LIN {X 0,Y 369.118,Z 198.507,A -85,B 0,C 180,E1 -12878.761,E2 -12878.761} C_VEL
LIN {X 0,Y 369.001,Z 198.517,A -85,B 0,C 180,E1 -12882.092,E2 -12882.092} C_VEL
LIN {X 0,Y 368.993,Z 198.519,A -85,B 0,C 180,E1 -12885.453,E2 -12885.453} C_VEL
LIN {X 0,Y 368.349,Z 198.603,A -85,B 0,C 180,E1 -12886.364,E2 -12886.364} C_VEL
LIN {X 0,Y 365.461,Z 198.96,A -85,B 0,C 180,E1 -12887.844,E2 -12887.844} C_VEL
LIN {X 0,Y 363.003,Z 199.268,A -85,B 0,C 180,E1 -12889.041,E2 -12889.041} C_VEL
LIN {X 0,Y 361.96,Z 199.395,A -85,B 0,C 180,E1 -12889.968,E2 -12889.968} C_VEL
LIN {X 0,Y 361.883,Z 199.405,A -85,B 0,C 180,E1 -12890.282,E2 -12890.282} C_VEL
LIN {X 0,Y 361.89,Z 199.404,A -85,B 0,C 180,E1 -12894.113,E2 -12894.113} C_VEL
LIN {X 0,Y 361.937,Z 199.403,A -85,B 0,C 180,E1 -12896.721,E2 -12896.721} C_VEL
LIN {X 0,Y 361.868,Z 199.409,A -85,B 0,C 180,E1 -12900.327,E2 -12900.327} C_VEL
LIN {X 0,Y 361.854,Z 199.411,A -85,B 0,C 180,E1 -12904.279,E2 -12904.279} C_VEL
LIN {X 0,Y 361.859,Z 199.407,A -85,B 0,C 180,E1 -12907.223,E2 -12907.223} C_VEL
LIN {X 0,Y 361.899,Z 199.405,A -85,B 0,C 180,E1 -12910.768,E2 -12910.768} C_VEL
LIN {X 0,Y 361.896,Z 199.408,A -85,B 0,C 180,E1 -12914.355,E2 -12914.355} C_VEL
LIN {X 0,Y 361.849,Z 199.408,A -85,B 0,C 180,E1 -12917.564,E2 -12917.564} C_VEL
LIN {X 0,Y 361.866,Z 199.406,A -85,B 0,C 180,E1 -12920.972,E2 -12920.972} C_VEL
LIN {X 0,Y 361.866,Z 199.408,A -85,B 0,C 180,E1 -12924.655,E2 -12924.655} C_VEL
LIN {X 0,Y 361.853,Z 199.412,A -85,B 0,C 180,E1 -12928.373,E2 -12928.373} C_VEL
LIN {X 0,Y 361.915,Z 199.405,A -85,B 0,C 180,E1 -12932.222,E2 -12932.222} C_VEL
LIN {X 0,Y 361.92,Z 199.4,A -85,B 0,C 180,E1 -12934.71,E2 -12934.71} C_VEL
LIN {X 0,Y 361.883,Z 199.407,A -85,B 0,C 180,E1 -12938.347,E2 -12938.347} C_VEL
LIN {X 0,Y 361.959,Z 199.4,A -85,B 0,C 180,E1 -12942.061,E2 -12942.061} C_VEL
LIN {X 0,Y 361.989,Z 199.395,A -85,B 0,C 180,E1 -12946.101,E2 -12946.101} C_VEL
LIN {X 0,Y 362.023,Z 199.392,A -85,B 0,C 180,E1 -12949.938,E2 -12949.938} C_VEL
LIN {X 0,Y 362.154,Z 199.372,A -85,B 0,C 180,E1 -12953.314,E2 -12953.314} C_VEL
LIN {X 0,Y 362.272,Z 199.361,A -85,B 0,C 180,E1 -12957.777,E2 -12957.777} C_VEL
LIN {X 0,Y 362.42,Z 199.34,A -85,B 0,C 180,E1 -12960.001,E2 -12960.001} C_VEL
LIN {X 0,Y 362.273,Z 199.356,A -85,B 0,C 180,E1 -12962.224,E2 -12962.224} C_VEL
LIN {X 0,Y 362.163,Z 199.369,A -85,B 0,C 180,E1 -12966.687,E2 -12966.687} C_VEL
LIN {X 0,Y 362.067,Z 199.382,A -85,B 0,C 180,E1 -12968.934,E2 -12968.934} C_VEL
LIN {X 0,Y 361.953,Z 199.395,A -85,B 0,C 180,E1 -12972.333,E2 -12972.333} C_VEL
LIN {X 0,Y 361.955,Z 199.395,A -85,B 0,C 180,E1 -12974.621,E2 -12974.621} C_VEL
LIN {X 0,Y 361.949,Z 199.396,A -85,B 0,C 180,E1 -12978.1,E2 -12978.1} C_VEL
LIN {X 0,Y 361.887,Z 199.406,A -85,B 0,C 180,E1 -12981.654,E2 -12981.654} C_VEL
LIN {X 0,Y 361.923,Z 199.405,A -85,B 0,C 180,E1 -12985.291,E2 -12985.291} C_VEL
LIN {X 0,Y 361.903,Z 199.403,A -85,B 0,C 180,E1 -12987.78,E2 -12987.78} C_VEL
LIN {X 0,Y 361.832,Z 199.412,A -85,B 0,C 180,E1 -12991.63,E2 -12991.63} C_VEL
LIN {X 0,Y 361.869,Z 199.409,A -85,B 0,C 180,E1 -12995.346,E2 -12995.346} C_VEL
LIN {X 0,Y 361.865,Z 199.412,A -85,B 0,C 180,E1 -12999.028,E2 -12999.028} C_VEL
LIN {X 0,Y 361.832,Z 199.415,A -85,B 0,C 180,E1 -13002.83,E2 -13002.83} C_VEL
LIN {X 0,Y 361.814,Z 199.412,A -85,B 0,C 180,E1 -13005.948,E2 -13005.948} C_VEL
LIN {X 0,Y 361.832,Z 199.413,A -85,B 0,C 180,E1 -13009.246,E2 -13009.246} C_VEL
LIN {X 0,Y 361.861,Z 199.412,A -85,B 0,C 180,E1 -13012.779,E2 -13012.779} C_VEL
LIN {X 0,Y 361.853,Z 199.412,A -85,B 0,C 180,E1 -13015.721,E2 -13015.721} C_VEL
LIN {X 0,Y 361.922,Z 199.576,A -85,B 0,C 180,E1 -13018.36,E2 -13018.36} C_VEL
LIN {X 0,Y 366.088,Z 217.855,A -85,B 0,C 180,E1 -13022.018,E2 -13022.018} C_VEL
LIN {X 0,Y 367.272,Z 224.486,A -85,B 0,C 180,E1 -13023.277,E2 -13023.277} C_VEL
LIN {X 0,Y 365.521,Z 242.961,A -85,B 0,C 180,E1 -13026.487,E2 -13026.487} C_VEL
LIN {X 0,Y 364.027,Z 261.035,A -85,B 0,C 180,E1 -13029.592,E2 -13029.592} C_VEL
LIN {X 0,Y 364.567,Z 267.895,A -85,B 0,C 180,E1 -13029.815,E2 -13029.815} C_VEL
LIN {X 0,Y 366.923,Z 292.032,A -85,B 0,C 180,E1 -13030.464,E2 -13030.464} C_VEL
LIN {X 0,Y 365.654,Z 367.753,A -85,B 0,C 180,E1 -13032.163,E2 -13032.163} C_VEL
LIN {X 0,Y 365.071,Z 380.038,A -85,B 0,C 180,E1 -13032.64,E2 -13032.64} C_VEL
LIN {X 0,Y 364.412,Z 392.244,A -85,B 0,C 180,E1 -13033.33,E2 -13033.33} C_VEL
LIN {X 0,Y 363.594,Z 404.788,A -85,B 0,C 180,E1 -13034.3,E2 -13034.3} C_VEL
LIN {X 0,Y 362.777,Z 415.954,A -85,B 0,C 180,E1 -13035.414,E2 -13035.414} C_VEL
LIN {X 0,Y 362.223,Z 424.979,A -85,B 0,C 180,E1 -13036.537,E2 -13036.537} C_VEL
LIN {X 0,Y 361.507,Z 434.174,A -85,B 0,C 180,E1 -13037.938,E2 -13037.938} C_VEL
LIN {X 0,Y 361.008,Z 443.11,A -85,B 0,C 180,E1 -13039.627,E2 -13039.627} C_VEL
LIN {X 0,Y 360.768,Z 450.158,A -85,B 0,C 180,E1 -13041.317,E2 -13041.317} C_VEL
LIN {X 0,Y 360.739,Z 456.564,A -85,B 0,C 180,E1 -13043.288,E2 -13043.288} C_VEL
LIN {X 0,Y 360.684,Z 460.629,A -85,B 0,C 180,E1 -13044.97,E2 -13044.97} C_VEL
LIN {X 0,Y 360.827,Z 463.562,A -85,B 0,C 180,E1 -13046.651,E2 -13046.651} C_VEL
LIN {X 0,Y 360.942,Z 464.906,A -85,B 0,C 180,E1 -13047.769,E2 -13047.769} C_VEL
LIN {X 0,Y 360.853,Z 465.795,A -85,B 0,C 180,E1 -13048.885,E2 -13048.885} C_VEL
LIN {X 0,Y 360.828,Z 466.258,A -85,B 0,C 180,E1 -13050.001,E2 -13050.001} C_VEL
LIN {X 0,Y 360.849,Z 466.244,A -85,B 0,C 180,E1 -13051.117,E2 -13051.117} C_VEL
LIN {X 0,Y 360.809,Z 465.799,A -85,B 0,C 180,E1 -13052.233,E2 -13052.233} C_VEL
LIN {X 0,Y 360.728,Z 464.934,A -85,B 0,C 180,E1 -13053.352,E2 -13053.352} C_VEL
LIN {X 0,Y 360.603,Z 463.587,A -85,B 0,C 180,E1 -13054.472,E2 -13054.472} C_VEL
LIN {X 0,Y 360.614,Z 460.433,A -85,B 0,C 180,E1 -13056.308,E2 -13056.308} C_VEL
LIN {X 0,Y 360.671,Z 456.84,A -85,B 0,C 180,E1 -13057.84,E2 -13057.84} C_VEL
LIN {X 0,Y 360.843,Z 451.756,A -85,B 0,C 180,E1 -13059.53,E2 -13059.53} C_VEL
LIN {X 0,Y 361.284,Z 445.363,A -85,B 0,C 180,E1 -13061.218,E2 -13061.218} C_VEL
LIN {X 0,Y 362.058,Z 437.426,A -85,B 0,C 180,E1 -13062.899,E2 -13062.899} C_VEL
LIN {X 0,Y 362.963,Z 429.132,A -85,B 0,C 180,E1 -13064.318,E2 -13064.318} C_VEL
LIN {X 0,Y 364.091,Z 418.285,A -85,B 0,C 180,E1 -13065.823,E2 -13065.823} C_VEL
LIN {X 0,Y 365.254,Z 408.426,A -85,B 0,C 180,E1 -13066.92,E2 -13066.92} C_VEL
LIN {X 0,Y 366.553,Z 395.984,A -85,B 0,C 180,E1 -13068.01,E2 -13068.01} C_VEL
LIN {X 0,Y 367.703,Z 383.82,A -85,B 0,C 180,E1 -13068.817,E2 -13068.817} C_VEL
LIN {X 0,Y 368.675,Z 370.254,A -85,B 0,C 180,E1 -13069.452,E2 -13069.452} C_VEL
LIN {X 0,Y 369.241,Z 356.669,A -85,B 0,C 180,E1 -13069.855,E2 -13069.855} C_VEL
LIN {X 0,Y 370.878,Z 292.289,A -85,B 0,C 180,E1 -13071.366,E2 -13071.366} C_VEL
LIN {X 0,Y 368.918,Z 273.49,A -85,B 0,C 180,E1 -13072.034,E2 -13072.034} C_VEL
LIN {X 0,Y 366.562,Z 258.445,A -85,B 0,C 180,E1 -13072.665,E2 -13072.665} C_VEL
LIN {X 0,Y 368.887,Z 236.241,A -85,B 0,C 180,E1 -13076.434,E2 -13076.434} C_VEL
LIN {X 0,Y 369.664,Z 228.641,A -85,B 0,C 180,E1 -13077.762,E2 -13077.762} C_VEL
LIN {X 0,Y 367.627,Z 218.97,A -85,B 0,C 180,E1 -13079.805,E2 -13079.805} C_VEL
LIN {X 0,Y 364.549,Z 207.813,A -85,B 0,C 180,E1 -13082.388,E2 -13082.388} C_VEL
LIN {X 0,Y 361.903,Z 199.531,A -85,B 0,C 180,E1 -13084.55,E2 -13084.55} C_VEL
LIN {X 0,Y 361.846,Z 199.412,A -85,B 0,C 180,E1 -13088.428,E2 -13088.428} C_VEL
LIN {X 0,Y 361.833,Z 199.413,A -85,B 0,C 180,E1 -13092.431,E2 -13092.431} C_VEL
LIN {X 0,Y 361.821,Z 199.413,A -85,B 0,C 180,E1 -13095.947,E2 -13095.947} C_VEL
LIN {X 0,Y 361.838,Z 199.413,A -85,B 0,C 180,E1 -13099.245,E2 -13099.245} C_VEL
LIN {X 0,Y 361.866,Z 199.409,A -85,B 0,C 180,E1 -13102.777,E2 -13102.777} C_VEL
LIN {X 0,Y 361.857,Z 199.409,A -85,B 0,C 180,E1 -13105.719,E2 -13105.719} C_VEL
LIN {X 0,Y 361.876,Z 199.408,A -85,B 0,C 180,E1 -13109.672,E2 -13109.672} C_VEL
LIN {X 0,Y 361.957,Z 199.397,A -85,B 0,C 180,E1 -13113.475,E2 -13113.475} C_VEL
LIN {X 0,Y 361.893,Z 199.403,A -85,B 0,C 180,E1 -13117.144,E2 -13117.144} C_VEL
LIN {X 0,Y 361.909,Z 199.403,A -85,B 0,C 180,E1 -13120.723,E2 -13120.723} C_VEL
LIN {X 0,Y 361.935,Z 199.401,A -85,B 0,C 180,E1 -13123.066,E2 -13123.066} C_VEL
LIN {X 0,Y 362.001,Z 199.394,A -85,B 0,C 180,E1 -13126.527,E2 -13126.527} C_VEL
LIN {X 0,Y 362.002,Z 199.394,A -85,B 0,C 180,E1 -13129.937,E2 -13129.937} C_VEL
LIN {X 0,Y 362.127,Z 199.581,A -85,B 0,C 180,E1 -13132.192,E2 -13132.192} C_VEL
LIN {X 0,Y 364.475,Z 207.695,A -85,B 0,C 180,E1 -13134.467,E2 -13134.467} C_VEL
LIN {X 0,Y 367.073,Z 217.573,A -85,B 0,C 180,E1 -13137.04,E2 -13137.04} C_VEL
LIN {X 0,Y 367.388,Z 220.859,A -85,B 0,C 180,E1 -13137.807,E2 -13137.807} C_VEL
LIN {X 0,Y 366.614,Z 232.738,A -85,B 0,C 180,E1 -13140.311,E2 -13140.311} C_VEL
LIN {X 0,Y 370.37,Z 248.389,A -85,B 0,C 180,E1 -13141.153,E2 -13141.153} C_VEL
LIN {X 0,Y 371.438,Z 253.878,A -85,B 0,C 180,E1 -13141.414,E2 -13141.414} C_VEL
LIN {X 0,Y 369.117,Z 317.897,A -85,B 0,C 180,E1 -13143.206,E2 -13143.206} C_VEL
LIN {X 0,Y 368.661,Z 330.151,A -85,B 0,C 180,E1 -13143.757,E2 -13143.757} C_VEL
LIN {X 0,Y 367.891,Z 342.582,A -85,B 0,C 180,E1 -13144.567,E2 -13144.567} C_VEL
LIN {X 0,Y 367.075,Z 353.098,A -85,B 0,C 180,E1 -13145.493,E2 -13145.493} C_VEL
LIN {X 0,Y 366.125,Z 363.059,A -85,B 0,C 180,E1 -13146.613,E2 -13146.613} C_VEL
LIN {X 0,Y 365.122,Z 372.767,A -85,B 0,C 180,E1 -13148.021,E2 -13148.021} C_VEL
LIN {X 0,Y 364.273,Z 379.966,A -85,B 0,C 180,E1 -13149.347,E2 -13149.347} C_VEL
LIN {X 0,Y 363.412,Z 386.564,A -85,B 0,C 180,E1 -13150.868,E2 -13150.868} C_VEL
LIN {X 0,Y 362.746,Z 391.42,A -85,B 0,C 180,E1 -13152.305,E2 -13152.305} C_VEL
LIN {X 0,Y 362.112,Z 395.64,A -85,B 0,C 180,E1 -13153.971,E2 -13153.971} C_VEL
LIN {X 0,Y 361.583,Z 398.748,A -85,B 0,C 180,E1 -13155.79,E2 -13155.79} C_VEL
LIN {X 0,Y 361.22,Z 400.374,A -85,B 0,C 180,E1 -13157.568,E2 -13157.568} C_VEL
LIN {X 0,Y 361.004,Z 400.698,A -85,B 0,C 180,E1 -13159.326,E2 -13159.326} C_VEL
LIN {X 0,Y 360.924,Z 399.948,A -85,B 0,C 180,E1 -13160.825,E2 -13160.825} C_VEL
LIN {X 0,Y 360.93,Z 399.056,A -85,B 0,C 180,E1 -13161.713,E2 -13161.713} C_VEL
LIN {X 0,Y 361.009,Z 397.344,A -85,B 0,C 180,E1 -13162.914,E2 -13162.914} C_VEL
LIN {X 0,Y 361.224,Z 393.503,A -85,B 0,C 180,E1 -13164.727,E2 -13164.727} C_VEL
LIN {X 0,Y 361.586,Z 387.777,A -85,B 0,C 180,E1 -13166.609,E2 -13166.609} C_VEL
LIN {X 0,Y 361.901,Z 381.824,A -85,B 0,C 180,E1 -13168.094,E2 -13168.094} C_VEL
LIN {X 0,Y 362.441,Z 373.721,A -85,B 0,C 180,E1 -13169.669,E2 -13169.669} C_VEL
LIN {X 0,Y 362.996,Z 364.815,A -85,B 0,C 180,E1 -13171.029,E2 -13171.029} C_VEL
LIN {X 0,Y 363.509,Z 355.694,A -85,B 0,C 180,E1 -13172.147,E2 -13172.147} C_VEL
LIN {X 0,Y 364.102,Z 344.601,A -85,B 0,C 180,E1 -13173.209,E2 -13173.209} C_VEL
LIN {X 0,Y 364.55,Z 332.719,A -85,B 0,C 180,E1 -13174.066,E2 -13174.066} C_VEL
LIN {X 0,Y 364.913,Z 321.208,A -85,B 0,C 180,E1 -13174.662,E2 -13174.662} C_VEL
LIN {X 0,Y 365.142,Z 308.779,A -85,B 0,C 180,E1 -13175.079,E2 -13175.079} C_VEL
LIN {X 0,Y 366.241,Z 249.047,A -85,B 0,C 180,E1 -13176.541,E2 -13176.541} C_VEL
LIN {X 0,Y 363.319,Z 230.123,A -85,B 0,C 180,E1 -13177.174,E2 -13177.174} C_VEL
LIN {X 0,Y 363.83,Z 216.259,A -85,B 0,C 180,E1 -13180.323,E2 -13180.323} C_VEL
LIN {X 0,Y 364.006,Z 210.426,A -85,B 0,C 180,E1 -13181.686,E2 -13181.686} C_VEL
LIN {X 0,Y 361.885,Z 199.568,A -85,B 0,C 180,E1 -13184.454,E2 -13184.454} C_VEL
LIN {X 0,Y 361.835,Z 199.415,A -85,B 0,C 180,E1 -13187.567,E2 -13187.567} C_VEL
LIN {X 0,Y 361.867,Z 199.406,A -85,B 0,C 180,E1 -13190.973,E2 -13190.973} C_VEL
LIN {X 0,Y 361.873,Z 199.405,A -85,B 0,C 180,E1 -13194.655,E2 -13194.655} C_VEL
LIN {X 0,Y 361.838,Z 199.41,A -85,B 0,C 180,E1 -13198.37,E2 -13198.37} C_VEL
LIN {X 0,Y 361.899,Z 199.403,A -85,B 0,C 180,E1 -13200.955,E2 -13200.955} C_VEL
LIN {X 0,Y 361.953,Z 199.401,A -85,B 0,C 180,E1 -13203.474,E2 -13203.474} C_VEL
LIN {X 0,Y 361.889,Z 199.406,A -85,B 0,C 180,E1 -13207.144,E2 -13207.144} C_VEL
LIN {X 0,Y 361.919,Z 199.4,A -85,B 0,C 180,E1 -13210.723,E2 -13210.723} C_VEL
LIN {X 0,Y 361.944,Z 199.396,A -85,B 0,C 180,E1 -13214.225,E2 -13214.225} C_VEL
LIN {X 0,Y 361.997,Z 199.39,A -85,B 0,C 180,E1 -13216.527,E2 -13216.527} C_VEL
LIN {X 0,Y 362.029,Z 199.386,A -85,B 0,C 180,E1 -13219.937,E2 -13219.937} C_VEL
LIN {X 0,Y 362.149,Z 199.371,A -85,B 0,C 180,E1 -13222.192,E2 -13222.192} C_VEL
LIN {X 0,Y 362.116,Z 199.375,A -85,B 0,C 180,E1 -13224.43,E2 -13224.43} C_VEL
LIN {X 0,Y 362.28,Z 199.355,A -85,B 0,C 180,E1 -13227.776,E2 -13227.776} C_VEL
LIN {X 0,Y 362.425,Z 199.336,A -85,B 0,C 180,E1 -13229.999,E2 -13229.999} C_VEL
LIN {X 0,Y 362.28,Z 199.354,A -85,B 0,C 180,E1 -13232.223,E2 -13232.223} C_VEL
LIN {X 0,Y 362.157,Z 199.373,A -85,B 0,C 180,E1 -13236.686,E2 -13236.686} C_VEL
LIN {X 0,Y 362.028,Z 199.386,A -85,B 0,C 180,E1 -13240.061,E2 -13240.061} C_VEL
LIN {X 0,Y 361.993,Z 199.39,A -85,B 0,C 180,E1 -13243.898,E2 -13243.898} C_VEL
LIN {X 0,Y 361.962,Z 199.394,A -85,B 0,C 180,E1 -13247.938,E2 -13247.938} C_VEL
LIN {X 0,Y 361.883,Z 199.405,A -85,B 0,C 180,E1 -13250.282,E2 -13250.282} C_VEL
LIN {X 0,Y 361.233,Z 199.492,A -85,B 0,C 180,E1 -13251.211,E2 -13251.211} C_VEL
LIN {X 0,Y 358.371,Z 199.85,A -85,B 0,C 180,E1 -13252.722,E2 -13252.722} C_VEL
LIN {X 0,Y 355.949,Z 200.148,A -85,B 0,C 180,E1 -13253.944,E2 -13253.944} C_VEL
LIN {X 0,Y 354.927,Z 200.274,A -85,B 0,C 180,E1 -13254.89,E2 -13254.89} C_VEL
LIN {X 0,Y 354.854,Z 200.279,A -85,B 0,C 180,E1 -13255.211,E2 -13255.211} C_VEL
LIN {X 0,Y 354.845,Z 200.284,A -85,B 0,C 180,E1 -13258.38,E2 -13258.38} C_VEL
LIN {X 0,Y 354.787,Z 200.288,A -85,B 0,C 180,E1 -13261.594,E2 -13261.594} C_VEL
LIN {X 0,Y 354.81,Z 200.286,A -85,B 0,C 180,E1 -13265.058,E2 -13265.058} C_VEL
LIN {X 0,Y 354.801,Z 200.287,A -85,B 0,C 180,E1 -13267.882,E2 -13267.882} C_VEL
LIN {X 0,Y 354.833,Z 200.282,A -85,B 0,C 180,E1 -13271.181,E2 -13271.181} C_VEL
LIN {X 0,Y 354.85,Z 200.285,A -85,B 0,C 180,E1 -13274.521,E2 -13274.521} C_VEL
LIN {X 0,Y 354.806,Z 200.286,A -85,B 0,C 180,E1 -13277.665,E2 -13277.665} C_VEL
LIN {X 0,Y 354.829,Z 200.285,A -85,B 0,C 180,E1 -13280.669,E2 -13280.669} C_VEL
LIN {X 0,Y 354.814,Z 200.29,A -85,B 0,C 180,E1 -13284.3,E2 -13284.3} C_VEL
LIN {X 0,Y 354.791,Z 200.289,A -85,B 0,C 180,E1 -13287.668,E2 -13287.668} C_VEL
LIN {X 0,Y 354.861,Z 200.28,A -85,B 0,C 180,E1 -13290.621,E2 -13290.621} C_VEL
LIN {X 0,Y 354.891,Z 200.28,A -85,B 0,C 180,E1 -13294.173,E2 -13294.173} C_VEL
LIN {X 0,Y 354.826,Z 200.288,A -85,B 0,C 180,E1 -13297.894,E2 -13297.894} C_VEL
LIN {X 0,Y 354.915,Z 200.277,A -85,B 0,C 180,E1 -13301.891,E2 -13301.891} C_VEL
LIN {X 0,Y 354.935,Z 200.275,A -85,B 0,C 180,E1 -13305.981,E2 -13305.981} C_VEL
LIN {X 0,Y 354.97,Z 200.27,A -85,B 0,C 180,E1 -13309.736,E2 -13309.736} C_VEL
LIN {X 0,Y 355.118,Z 200.247,A -85,B 0,C 180,E1 -13313.181,E2 -13313.181} C_VEL
LIN {X 0,Y 355.235,Z 200.238,A -85,B 0,C 180,E1 -13317.733,E2 -13317.733} C_VEL
LIN {X 0,Y 355.389,Z 200.216,A -85,B 0,C 180,E1 -13320.001,E2 -13320.001} C_VEL
LIN {X 0,Y 355.236,Z 200.233,A -85,B 0,C 180,E1 -13322.268,E2 -13322.268} C_VEL
LIN {X 0,Y 355.129,Z 200.245,A -85,B 0,C 180,E1 -13326.82,E2 -13326.82} C_VEL
LIN {X 0,Y 355.008,Z 200.262,A -85,B 0,C 180,E1 -13329.113,E2 -13329.113} C_VEL
LIN {X 0,Y 354.914,Z 200.272,A -85,B 0,C 180,E1 -13332.582,E2 -13332.582} C_VEL
LIN {X 0,Y 354.883,Z 200.276,A -85,B 0,C 180,E1 -13336.097,E2 -13336.097} C_VEL
LIN {X 0,Y 354.895,Z 200.274,A -85,B 0,C 180,E1 -13338.473,E2 -13338.473} C_VEL
LIN {X 0,Y 354.83,Z 200.283,A -85,B 0,C 180,E1 -13342.107,E2 -13342.107} C_VEL
LIN {X 0,Y 354.893,Z 200.276,A -85,B 0,C 180,E1 -13345.828,E2 -13345.828} C_VEL
LIN {X 0,Y 354.812,Z 200.286,A -85,B 0,C 180,E1 -13349.683,E2 -13349.683} C_VEL
LIN {X 0,Y 354.801,Z 200.287,A -85,B 0,C 180,E1 -13353.703,E2 -13353.703} C_VEL
LIN {X 0,Y 354.793,Z 200.288,A -85,B 0,C 180,E1 -13356.461,E2 -13356.461} C_VEL
LIN {X 0,Y 354.82,Z 200.286,A -85,B 0,C 180,E1 -13359.425,E2 -13359.425} C_VEL
LIN {X 0,Y 354.784,Z 200.293,A -85,B 0,C 180,E1 -13362.868,E2 -13362.868} C_VEL
LIN {X 0,Y 354.763,Z 200.291,A -85,B 0,C 180,E1 -13366.105,E2 -13366.105} C_VEL
LIN {X 0,Y 354.784,Z 200.291,A -85,B 0,C 180,E1 -13369.18,E2 -13369.18} C_VEL
LIN {X 0,Y 354.804,Z 200.287,A -85,B 0,C 180,E1 -13372.404,E2 -13372.404} C_VEL
LIN {X 0,Y 354.81,Z 200.291,A -85,B 0,C 180,E1 -13374.942,E2 -13374.942} C_VEL
LIN {X 0,Y 354.864,Z 200.477,A -85,B 0,C 180,E1 -13378.052,E2 -13378.052} C_VEL
LIN {X 0,Y 359.007,Z 218.586,A -85,B 0,C 180,E1 -13381.756,E2 -13381.756} C_VEL
LIN {X 0,Y 360.296,Z 225.133,A -85,B 0,C 180,E1 -13383.032,E2 -13383.032} C_VEL
LIN {X 0,Y 359.033,Z 238.587,A -85,B 0,C 180,E1 -13385.421,E2 -13385.421} C_VEL
LIN {X 0,Y 357.085,Z 260.763,A -85,B 0,C 180,E1 -13389.319,E2 -13389.319} C_VEL
LIN {X 0,Y 358.098,Z 273.042,A -85,B 0,C 180,E1 -13389.692,E2 -13389.692} C_VEL
LIN {X 0,Y 359.973,Z 293.475,A -85,B 0,C 180,E1 -13390.248,E2 -13390.248} C_VEL
LIN {X 0,Y 358.736,Z 366.518,A -85,B 0,C 180,E1 -13391.918,E2 -13391.918} C_VEL
LIN {X 0,Y 358.104,Z 379.758,A -85,B 0,C 180,E1 -13392.439,E2 -13392.439} C_VEL
LIN {X 0,Y 357.408,Z 391.868,A -85,B 0,C 180,E1 -13393.141,E2 -13393.141} C_VEL
LIN {X 0,Y 356.591,Z 404.377,A -85,B 0,C 180,E1 -13394.131,E2 -13394.131} C_VEL
LIN {X 0,Y 355.788,Z 415.287,A -85,B 0,C 180,E1 -13395.241,E2 -13395.241} C_VEL
LIN {X 0,Y 355.164,Z 424.502,A -85,B 0,C 180,E1 -13396.41,E2 -13396.41} C_VEL
LIN {X 0,Y 354.4,Z 434.514,A -85,B 0,C 180,E1 -13397.983,E2 -13397.983} C_VEL
LIN {X 0,Y 353.971,Z 441.921,A -85,B 0,C 180,E1 -13399.418,E2 -13399.418} C_VEL
LIN {X 0,Y 353.683,Z 449.1,A -85,B 0,C 180,E1 -13401.142,E2 -13401.142} C_VEL
LIN {X 0,Y 353.673,Z 453.943,A -85,B 0,C 180,E1 -13402.58,E2 -13402.58} C_VEL
LIN {X 0,Y 353.694,Z 458.499,A -85,B 0,C 180,E1 -13404.299,E2 -13404.299} C_VEL
LIN {X 0,Y 353.598,Z 460.845,A -85,B 0,C 180,E1 -13405.441,E2 -13405.441} C_VEL
LIN {X 0,Y 353.761,Z 462.754,A -85,B 0,C 180,E1 -13406.584,E2 -13406.584} C_VEL
LIN {X 0,Y 353.893,Z 464.14,A -85,B 0,C 180,E1 -13407.725,E2 -13407.725} C_VEL
LIN {X 0,Y 353.808,Z 465.058,A -85,B 0,C 180,E1 -13408.863,E2 -13408.863} C_VEL
LIN {X 0,Y 353.78,Z 465.554,A -85,B 0,C 180,E1 -13410.001,E2 -13410.001} C_VEL
LIN {X 0,Y 353.8,Z 465.581,A -85,B 0,C 180,E1 -13411.139,E2 -13411.139} C_VEL
LIN {X 0,Y 353.737,Z 465.159,A -85,B 0,C 180,E1 -13412.278,E2 -13412.278} C_VEL
LIN {X 0,Y 353.632,Z 464.317,A -85,B 0,C 180,E1 -13413.419,E2 -13413.419} C_VEL
LIN {X 0,Y 353.526,Z 463.026,A -85,B 0,C 180,E1 -13414.562,E2 -13414.562} C_VEL
LIN {X 0,Y 353.518,Z 460.257,A -85,B 0,C 180,E1 -13416.271,E2 -13416.271} C_VEL
LIN {X 0,Y 353.571,Z 456.381,A -85,B 0,C 180,E1 -13417.999,E2 -13417.999} C_VEL
LIN {X 0,Y 353.787,Z 451.35,A -85,B 0,C 180,E1 -13419.722,E2 -13419.722} C_VEL
LIN {X 0,Y 354.292,Z 445.009,A -85,B 0,C 180,E1 -13421.442,E2 -13421.442} C_VEL
LIN {X 0,Y 355.085,Z 437.16,A -85,B 0,C 180,E1 -13423.157,E2 -13423.157} C_VEL
LIN {X 0,Y 356.144,Z 427.942,A -85,B 0,C 180,E1 -13424.771,E2 -13424.771} C_VEL
LIN {X 0,Y 357.25,Z 418.332,A -85,B 0,C 180,E1 -13426.134,E2 -13426.134} C_VEL
LIN {X 0,Y 358.494,Z 408.625,A -85,B 0,C 180,E1 -13427.249,E2 -13427.249} C_VEL
LIN {X 0,Y 359.685,Z 398.191,A -85,B 0,C 180,E1 -13428.218,E2 -13428.218} C_VEL
LIN {X 0,Y 360.894,Z 385.711,A -85,B 0,C 180,E1 -13429.112,E2 -13429.112} C_VEL
LIN {X 0,Y 361.962,Z 373.429,A -85,B 0,C 180,E1 -13429.754,E2 -13429.754} C_VEL
LIN {X 0,Y 362.61,Z 360.881,A -85,B 0,C 180,E1 -13430.197,E2 -13430.197} C_VEL
LIN {X 0,Y 364.548,Z 293.153,A -85,B 0,C 180,E1 -13431.846,E2 -13431.846} C_VEL
LIN {X 0,Y 362.577,Z 274.319,A -85,B 0,C 180,E1 -13432.535,E2 -13432.535} C_VEL
LIN {X 0,Y 360.02,Z 258.245,A -85,B 0,C 180,E1 -13433.232,E2 -13433.232} C_VEL
LIN {X 0,Y 362.35,Z 237.307,A -85,B 0,C 180,E1 -13436.848,E2 -13436.848} C_VEL
LIN {X 0,Y 363.076,Z 230.876,A -85,B 0,C 180,E1 -13437.993,E2 -13437.993} C_VEL
LIN {X 0,Y 361.091,Z 221.299,A -85,B 0,C 180,E1 -13440.078,E2 -13440.078} C_VEL
LIN {X 0,Y 358.056,Z 210.158,A -85,B 0,C 180,E1 -13442.745,E2 -13442.745} C_VEL
LIN {X 0,Y 354.865,Z 200.481,A -85,B 0,C 180,E1 -13445.373,E2 -13445.373} C_VEL
LIN {X 0,Y 354.797,Z 200.29,A -85,B 0,C 180,E1 -13447.884,E2 -13447.884} C_VEL
LIN {X 0,Y 354.774,Z 200.293,A -85,B 0,C 180,E1 -13451.168,E2 -13451.168} C_VEL
LIN {X 0,Y 354.766,Z 200.292,A -85,B 0,C 180,E1 -13454.506,E2 -13454.506} C_VEL
LIN {X 0,Y 354.797,Z 200.288,A -85,B 0,C 180,E1 -13457.662,E2 -13457.662} C_VEL
LIN {X 0,Y 354.819,Z 200.286,A -85,B 0,C 180,E1 -13460.666,E2 -13460.666} C_VEL
LIN {X 0,Y 354.825,Z 200.283,A -85,B 0,C 180,E1 -13464.301,E2 -13464.301} C_VEL
LIN {X 0,Y 354.79,Z 200.29,A -85,B 0,C 180,E1 -13467.666,E2 -13467.666} C_VEL
LIN {X 0,Y 354.85,Z 200.284,A -85,B 0,C 180,E1 -13471.618,E2 -13471.618} C_VEL
LIN {X 0,Y 354.902,Z 200.278,A -85,B 0,C 180,E1 -13474.172,E2 -13474.172} C_VEL
LIN {X 0,Y 354.838,Z 200.284,A -85,B 0,C 180,E1 -13477.894,E2 -13477.894} C_VEL
LIN {X 0,Y 354.925,Z 200.275,A -85,B 0,C 180,E1 -13481.891,E2 -13481.891} C_VEL
LIN {X 0,Y 354.945,Z 200.271,A -85,B 0,C 180,E1 -13485.981,E2 -13485.981} C_VEL
LIN {X 0,Y 354.958,Z 200.272,A -85,B 0,C 180,E1 -13489.735,E2 -13489.735} C_VEL
LIN {X 0,Y 355.062,Z 200.476,A -85,B 0,C 180,E1 -13491.348,E2 -13491.348} C_VEL
LIN {X 0,Y 357.879,Z 209.797,A -85,B 0,C 180,E1 -13494.082,E2 -13494.082} C_VEL
LIN {X 0,Y 360.579,Z 220.271,A -85,B 0,C 180,E1 -13496.887,E2 -13496.887} C_VEL
LIN {X 0,Y 360.761,Z 223.994,A -85,B 0,C 180,E1 -13497.767,E2 -13497.767} C_VEL
LIN {X 0,Y 360.124,Z 233.131,A -85,B 0,C 180,E1 -13499.72,E2 -13499.72} C_VEL
LIN {X 0,Y 363.944,Z 248.948,A -85,B 0,C 180,E1 -13500.622,E2 -13500.622} C_VEL
LIN {X 0,Y 365.125,Z 255.392,A -85,B 0,C 180,E1 -13500.93,E2 -13500.93} C_VEL
LIN {X 0,Y 362.685,Z 318.346,A -85,B 0,C 180,E1 -13502.741,E2 -13502.741} C_VEL
LIN {X 0,Y 362.171,Z 331.157,A -85,B 0,C 180,E1 -13503.337,E2 -13503.337} C_VEL
LIN {X 0,Y 361.453,Z 341.836,A -85,B 0,C 180,E1 -13504.041,E2 -13504.041} C_VEL
LIN {X 0,Y 360.535,Z 353.165,A -85,B 0,C 180,E1 -13505.03,E2 -13505.03} C_VEL
LIN {X 0,Y 359.568,Z 363.24,A -85,B 0,C 180,E1 -13506.171,E2 -13506.171} C_VEL
LIN {X 0,Y 358.673,Z 371.286,A -85,B 0,C 180,E1 -13507.317,E2 -13507.317} C_VEL
LIN {X 0,Y 357.637,Z 379.443,A -85,B 0,C 180,E1 -13508.759,E2 -13508.759} C_VEL
LIN {X 0,Y 356.747,Z 385.898,A -85,B 0,C 180,E1 -13510.212,E2 -13510.212} C_VEL
LIN {X 0,Y 355.869,Z 391.934,A -85,B 0,C 180,E1 -13511.967,E2 -13511.967} C_VEL
LIN {X 0,Y 355.182,Z 396.327,A -85,B 0,C 180,E1 -13513.735,E2 -13513.735} C_VEL
LIN {X 0,Y 354.768,Z 398.491,A -85,B 0,C 180,E1 -13514.923,E2 -13514.923} C_VEL
LIN {X 0,Y 354.463,Z 400.06,A -85,B 0,C 180,E1 -13516.115,E2 -13516.115} C_VEL
LIN {X 0,Y 354.136,Z 401.228,A -85,B 0,C 180,E1 -13517.714,E2 -13517.714} C_VEL
LIN {X 0,Y 353.899,Z 401.232,A -85,B 0,C 180,E1 -13519.73,E2 -13519.73} C_VEL
LIN {X 0,Y 353.847,Z 400.386,A -85,B 0,C 180,E1 -13521.012,E2 -13521.012} C_VEL
LIN {X 0,Y 353.939,Z 398.155,A -85,B 0,C 180,E1 -13522.78,E2 -13522.78} C_VEL
LIN {X 0,Y 354.159,Z 394.364,A -85,B 0,C 180,E1 -13524.627,E2 -13524.627} C_VEL
LIN {X 0,Y 354.474,Z 389.305,A -85,B 0,C 180,E1 -13526.374,E2 -13526.374} C_VEL
LIN {X 0,Y 354.818,Z 382.832,A -85,B 0,C 180,E1 -13528.061,E2 -13528.061} C_VEL
LIN {X 0,Y 355.347,Z 375.023,A -85,B 0,C 180,E1 -13529.633,E2 -13529.633} C_VEL
LIN {X 0,Y 355.912,Z 366.069,A -85,B 0,C 180,E1 -13531.055,E2 -13531.055} C_VEL
LIN {X 0,Y 356.526,Z 355.954,A -85,B 0,C 180,E1 -13532.323,E2 -13532.323} C_VEL
LIN {X 0,Y 357.136,Z 344.457,A -85,B 0,C 180,E1 -13533.435,E2 -13533.435} C_VEL
LIN {X 0,Y 357.609,Z 332.677,A -85,B 0,C 180,E1 -13534.288,E2 -13534.288} C_VEL
LIN {X 0,Y 357.945,Z 321.353,A -85,B 0,C 180,E1 -13534.878,E2 -13534.878} C_VEL
LIN {X 0,Y 358.183,Z 308.816,A -85,B 0,C 180,E1 -13535.303,E2 -13535.303} C_VEL
LIN {X 0,Y 359.3,Z 249.557,A -85,B 0,C 180,E1 -13536.79,E2 -13536.79} C_VEL
LIN {X 0,Y 356.372,Z 230.631,A -85,B 0,C 180,E1 -13537.413,E2 -13537.413} C_VEL
LIN {X 0,Y 356.673,Z 223.132,A -85,B 0,C 180,E1 -13539.089,E2 -13539.089} C_VEL
LIN {X 0,Y 357.1,Z 212.462,A -85,B 0,C 180,E1 -13541.593,E2 -13541.593} C_VEL
LIN {X 0,Y 355.151,Z 201.926,A -85,B 0,C 180,E1 -13544.263,E2 -13544.263} C_VEL
LIN {X 0,Y 354.823,Z 200.341,A -85,B 0,C 180,E1 -13544.753,E2 -13544.753} C_VEL
LIN {X 0,Y 354.793,Z 200.293,A -85,B 0,C 180,E1 -13547.662,E2 -13547.662} C_VEL
LIN {X 0,Y 354.814,Z 200.284,A -85,B 0,C 180,E1 -13550.665,E2 -13550.665} C_VEL
LIN {X 0,Y 354.82,Z 200.284,A -85,B 0,C 180,E1 -13554.3,E2 -13554.3} C_VEL
LIN {X 0,Y 354.788,Z 200.293,A -85,B 0,C 180,E1 -13557.666,E2 -13557.666} C_VEL
LIN {X 0,Y 354.867,Z 200.278,A -85,B 0,C 180,E1 -13560.621,E2 -13560.621} C_VEL
LIN {X 0,Y 354.898,Z 200.274,A -85,B 0,C 180,E1 -13564.172,E2 -13564.172} C_VEL
LIN {X 0,Y 354.833,Z 200.284,A -85,B 0,C 180,E1 -13567.893,E2 -13567.893} C_VEL
LIN {X 0,Y 354.921,Z 200.272,A -85,B 0,C 180,E1 -13571.891,E2 -13571.891} C_VEL
LIN {X 0,Y 354.941,Z 200.269,A -85,B 0,C 180,E1 -13575.98,E2 -13575.98} C_VEL
LIN {X 0,Y 354.976,Z 200.266,A -85,B 0,C 180,E1 -13579.735,E2 -13579.735} C_VEL
LIN {X 0,Y 355.112,Z 200.247,A -85,B 0,C 180,E1 -13582.036,E2 -13582.036} C_VEL
LIN {X 0,Y 355.091,Z 200.25,A -85,B 0,C 180,E1 -13584.32,E2 -13584.32} C_VEL
LIN {X 0,Y 355.243,Z 200.232,A -85,B 0,C 180,E1 -13587.732,E2 -13587.732} C_VEL
LIN {X 0,Y 355.395,Z 200.212,A -85,B 0,C 180,E1 -13589.999,E2 -13589.999} C_VEL
LIN {X 0,Y 355.243,Z 200.231,A -85,B 0,C 180,E1 -13592.267,E2 -13592.267} C_VEL
LIN {X 0,Y 355.122,Z 200.251,A -85,B 0,C 180,E1 -13596.819,E2 -13596.819} C_VEL
LIN {X 0,Y 354.974,Z 200.265,A -85,B 0,C 180,E1 -13600.263,E2 -13600.263} C_VEL
LIN {X 0,Y 354.938,Z 200.269,A -85,B 0,C 180,E1 -13604.018,E2 -13604.018} C_VEL
LIN {X 0,Y 354.918,Z 200.272,A -85,B 0,C 180,E1 -13608.108,E2 -13608.108} C_VEL
LIN {X 0,Y 354.83,Z 200.283,A -85,B 0,C 180,E1 -13612.105,E2 -13612.105} C_VEL
LIN {X 0,Y 354.854,Z 200.279,A -85,B 0,C 180,E1 -13615.211,E2 -13615.211} C_VEL
LIN {X 0,Y 354.214,Z 200.362,A -85,B 0,C 180,E1 -13616.157,E2 -13616.157} C_VEL
LIN {X 0,Y 351.364,Z 200.714,A -85,B 0,C 180,E1 -13617.696,E2 -13617.696} C_VEL
LIN {X 0,Y 348.922,Z 201.021,A -85,B 0,C 180,E1 -13618.942,E2 -13618.942} C_VEL
LIN {X 0,Y 347.856,Z 201.152,A -85,B 0,C 180,E1 -13619.906,E2 -13619.906} C_VEL
LIN {X 0,Y 347.762,Z 201.165,A -85,B 0,C 180,E1 -13620.233,E2 -13620.233} C_VEL
LIN {X 0,Y 347.742,Z 201.167,A -85,B 0,C 180,E1 -13624.043,E2 -13624.043} C_VEL
LIN {X 0,Y 347.757,Z 201.164,A -85,B 0,C 180,E1 -13627.32,E2 -13627.32} C_VEL
LIN {X 0,Y 347.787,Z 201.164,A -85,B 0,C 180,E1 -13630.288,E2 -13630.288} C_VEL
LIN {X 0,Y 347.776,Z 201.161,A -85,B 0,C 180,E1 -13633.398,E2 -13633.398} C_VEL
LIN {X 0,Y 347.762,Z 201.166,A -85,B 0,C 180,E1 -13636.678,E2 -13636.678} C_VEL
LIN {X 0,Y 347.75,Z 201.169,A -85,B 0,C 180,E1 -13640.171,E2 -13640.171} C_VEL
LIN {X 0,Y 347.758,Z 201.165,A -85,B 0,C 180,E1 -13642.68,E2 -13642.68} C_VEL
LIN {X 0,Y 347.74,Z 201.169,A -85,B 0,C 180,E1 -13645.956,E2 -13645.956} C_VEL
LIN {X 0,Y 347.764,Z 201.164,A -85,B 0,C 180,E1 -13649.654,E2 -13649.654} C_VEL
LIN {X 0,Y 347.823,Z 201.157,A -85,B 0,C 180,E1 -13653.608,E2 -13653.608} C_VEL
LIN {X 0,Y 347.78,Z 201.166,A -85,B 0,C 180,E1 -13656.162,E2 -13656.162} C_VEL
LIN {X 0,Y 347.809,Z 201.162,A -85,B 0,C 180,E1 -13659.91,E2 -13659.91} C_VEL
LIN {X 0,Y 347.859,Z 201.153,A -85,B 0,C 180,E1 -13662.359,E2 -13662.359} C_VEL
LIN {X 0,Y 347.889,Z 201.152,A -85,B 0,C 180,E1 -13665.971,E2 -13665.971} C_VEL
LIN {X 0,Y 347.921,Z 201.146,A -85,B 0,C 180,E1 -13669.526,E2 -13669.526} C_VEL
LIN {X 0,Y 348.084,Z 201.123,A -85,B 0,C 180,E1 -13673.042,E2 -13673.042} C_VEL
LIN {X 0,Y 348.198,Z 201.115,A -85,B 0,C 180,E1 -13677.687,E2 -13677.687} C_VEL
LIN {X 0,Y 348.338,Z 201.094,A -85,B 0,C 180,E1 -13680.001,E2 -13680.001} C_VEL
LIN {X 0,Y 348.198,Z 201.109,A -85,B 0,C 180,E1 -13682.314,E2 -13682.314} C_VEL
LIN {X 0,Y 348.098,Z 201.122,A -85,B 0,C 180,E1 -13686.958,E2 -13686.958} C_VEL
LIN {X 0,Y 347.96,Z 201.142,A -85,B 0,C 180,E1 -13689.299,E2 -13689.299} C_VEL
LIN {X 0,Y 347.883,Z 201.149,A -85,B 0,C 180,E1 -13692.84,E2 -13692.84} C_VEL
LIN {X 0,Y 347.832,Z 201.154,A -85,B 0,C 180,E1 -13696.432,E2 -13696.432} C_VEL
LIN {X 0,Y 347.845,Z 201.154,A -85,B 0,C 180,E1 -13698.861,E2 -13698.861} C_VEL
LIN {X 0,Y 347.769,Z 201.162,A -85,B 0,C 180,E1 -13702.58,E2 -13702.58} C_VEL
LIN {X 0,Y 347.807,Z 201.162,A -85,B 0,C 180,E1 -13705.109,E2 -13705.109} C_VEL
LIN {X 0,Y 347.803,Z 201.16,A -85,B 0,C 180,E1 -13707.695,E2 -13707.695} C_VEL
LIN {X 0,Y 347.744,Z 201.165,A -85,B 0,C 180,E1 -13710.349,E2 -13710.349} C_VEL
LIN {X 0,Y 347.744,Z 201.165,A -85,B 0,C 180,E1 -13714.045,E2 -13714.045} C_VEL
LIN {X 0,Y 347.757,Z 201.167,A -85,B 0,C 180,E1 -13717.322,E2 -13717.322} C_VEL
LIN {X 0,Y 347.728,Z 201.167,A -85,B 0,C 180,E1 -13720.298,E2 -13720.298} C_VEL
LIN {X 0,Y 347.719,Z 201.17,A -85,B 0,C 180,E1 -13723.409,E2 -13723.409} C_VEL
LIN {X 0,Y 347.722,Z 201.171,A -85,B 0,C 180,E1 -13726.688,E2 -13726.688} C_VEL
LIN {X 0,Y 347.744,Z 201.166,A -85,B 0,C 180,E1 -13730.174,E2 -13730.174} C_VEL
LIN {X 0,Y 347.759,Z 201.168,A -85,B 0,C 180,E1 -13732.68,E2 -13732.68} C_VEL
LIN {X 0,Y 347.747,Z 201.17,A -85,B 0,C 180,E1 -13735.957,E2 -13735.957} C_VEL
LIN {X 0,Y 347.827,Z 201.397,A -85,B 0,C 180,E1 -13737.745,E2 -13737.745} C_VEL
LIN {X 0,Y 351.767,Z 218.626,A -85,B 0,C 180,E1 -13741.349,E2 -13741.349} C_VEL
LIN {X 0,Y 353.25,Z 225.736,A -85,B 0,C 180,E1 -13742.769,E2 -13742.769} C_VEL
LIN {X 0,Y 352.826,Z 232.502,A -85,B 0,C 180,E1 -13744.011,E2 -13744.011} C_VEL
LIN {X 0,Y 350.526,Z 255.91,A -85,B 0,C 180,E1 -13748.229,E2 -13748.229} C_VEL
LIN {X 0,Y 350.153,Z 260.979,A -85,B 0,C 180,E1 -13749.076,E2 -13749.076} C_VEL
LIN {X 0,Y 353.071,Z 293.175,A -85,B 0,C 180,E1 -13749.986,E2 -13749.986} C_VEL
LIN {X 0,Y 351.782,Z 365.948,A -85,B 0,C 180,E1 -13751.699,E2 -13751.699} C_VEL
LIN {X 0,Y 351.141,Z 379.166,A -85,B 0,C 180,E1 -13752.229,E2 -13752.229} C_VEL
LIN {X 0,Y 350.417,Z 391.276,A -85,B 0,C 180,E1 -13752.944,E2 -13752.944} C_VEL
LIN {X 0,Y 349.591,Z 403.789,A -85,B 0,C 180,E1 -13753.954,E2 -13753.954} C_VEL
LIN {X 0,Y 348.741,Z 415.177,A -85,B 0,C 180,E1 -13755.143,E2 -13755.143} C_VEL
LIN {X 0,Y 348.099,Z 423.915,A -85,B 0,C 180,E1 -13756.278,E2 -13756.278} C_VEL
LIN {X 0,Y 347.383,Z 433.097,A -85,B 0,C 180,E1 -13757.736,E2 -13757.736} C_VEL
LIN {X 0,Y 346.929,Z 440.641,A -85,B 0,C 180,E1 -13759.201,E2 -13759.201} C_VEL
LIN {X 0,Y 346.615,Z 447.986,A -85,B 0,C 180,E1 -13760.96,E2 -13760.96} C_VEL
LIN {X 0,Y 346.604,Z 452.907,A -85,B 0,C 180,E1 -13762.427,E2 -13762.427} C_VEL
LIN {X 0,Y 346.635,Z 457.57,A -85,B 0,C 180,E1 -13764.183,E2 -13764.183} C_VEL
LIN {X 0,Y 346.535,Z 459.953,A -85,B 0,C 180,E1 -13765.348,E2 -13765.348} C_VEL
LIN {X 0,Y 346.697,Z 461.899,A -85,B 0,C 180,E1 -13766.514,E2 -13766.514} C_VEL
LIN {X 0,Y 346.826,Z 463.351,A -85,B 0,C 180,E1 -13767.678,E2 -13767.678} C_VEL
LIN {X 0,Y 346.763,Z 464.301,A -85,B 0,C 180,E1 -13768.84,E2 -13768.84} C_VEL
LIN {X 0,Y 346.732,Z 464.828,A -85,B 0,C 180,E1 -13770.001,E2 -13770.001} C_VEL
LIN {X 0,Y 346.752,Z 464.917,A -85,B 0,C 180,E1 -13771.162,E2 -13771.162} C_VEL
LIN {X 0,Y 346.665,Z 464.521,A -85,B 0,C 180,E1 -13772.325,E2 -13772.325} C_VEL
LIN {X 0,Y 346.537,Z 463.703,A -85,B 0,C 180,E1 -13773.489,E2 -13773.489} C_VEL
LIN {X 0,Y 346.45,Z 462.463,A -85,B 0,C 180,E1 -13774.655,E2 -13774.655} C_VEL
LIN {X 0,Y 346.44,Z 459.989,A -85,B 0,C 180,E1 -13776.26,E2 -13776.26} C_VEL
LIN {X 0,Y 346.502,Z 455.922,A -85,B 0,C 180,E1 -13778.163,E2 -13778.163} C_VEL
LIN {X 0,Y 346.724,Z 450.959,A -85,B 0,C 180,E1 -13779.922,E2 -13779.922} C_VEL
LIN {X 0,Y 347.313,Z 444.716,A -85,B 0,C 180,E1 -13781.675,E2 -13781.675} C_VEL
LIN {X 0,Y 348.122,Z 436.963,A -85,B 0,C 180,E1 -13783.425,E2 -13783.425} C_VEL
LIN {X 0,Y 349.161,Z 428.642,A -85,B 0,C 180,E1 -13784.947,E2 -13784.947} C_VEL
LIN {X 0,Y 350.43,Z 418.377,A -85,B 0,C 180,E1 -13786.457,E2 -13786.457} C_VEL
LIN {X 0,Y 351.933,Z 407.498,A -85,B 0,C 180,E1 -13787.731,E2 -13787.731} C_VEL
LIN {X 0,Y 353.33,Z 395.208,A -85,B 0,C 180,E1 -13788.859,E2 -13788.859} C_VEL
LIN {X 0,Y 354.573,Z 383.316,A -85,B 0,C 180,E1 -13789.692,E2 -13789.692} C_VEL
LIN {X 0,Y 355.678,Z 370.283,A -85,B 0,C 180,E1 -13790.344,E2 -13790.344} C_VEL
LIN {X 0,Y 356.367,Z 356.497,A -85,B 0,C 180,E1 -13790.793,E2 -13790.793} C_VEL
LIN {X 0,Y 358.2,Z 293.209,A -85,B 0,C 180,E1 -13792.372,E2 -13792.372} C_VEL
LIN {X 0,Y 356.266,Z 274.745,A -85,B 0,C 180,E1 -13793.078,E2 -13793.078} C_VEL
LIN {X 0,Y 353.518,Z 257.717,A -85,B 0,C 180,E1 -13793.866,E2 -13793.866} C_VEL
LIN {X 0,Y 355.856,Z 238.415,A -85,B 0,C 180,E1 -13797.285,E2 -13797.285} C_VEL
LIN {X 0,Y 356.51,Z 233.191,A -85,B 0,C 180,E1 -13798.238,E2 -13798.238} C_VEL
LIN {X 0,Y 354.593,Z 223.69,A -85,B 0,C 180,E1 -13800.359,E2 -13800.359} C_VEL
LIN {X 0,Y 351.748,Z 213.212,A -85,B 0,C 180,E1 -13802.947,E2 -13802.947} C_VEL
LIN {X 0,Y 348.933,Z 204.714,A -85,B 0,C 180,E1 -13805.296,E2 -13805.296} C_VEL
LIN {X 0,Y 347.779,Z 201.269,A -85,B 0,C 180,E1 -13806.384,E2 -13806.384} C_VEL
LIN {X 0,Y 347.704,Z 201.174,A -85,B 0,C 180,E1 -13809.818,E2 -13809.818} C_VEL
LIN {X 0,Y 347.728,Z 201.173,A -85,B 0,C 180,E1 -13813.313,E2 -13813.313} C_VEL
LIN {X 0,Y 347.728,Z 201.17,A -85,B 0,C 180,E1 -13816.686,E2 -13816.686} C_VEL
LIN {X 0,Y 347.75,Z 201.164,A -85,B 0,C 180,E1 -13820.173,E2 -13820.173} C_VEL
LIN {X 0,Y 347.764,Z 201.165,A -85,B 0,C 180,E1 -13822.679,E2 -13822.679} C_VEL
LIN {X 0,Y 347.752,Z 201.166,A -85,B 0,C 180,E1 -13825.956,E2 -13825.956} C_VEL
LIN {X 0,Y 347.752,Z 201.168,A -85,B 0,C 180,E1 -13829.652,E2 -13829.652} C_VEL
LIN {X 0,Y 347.834,Z 201.157,A -85,B 0,C 180,E1 -13833.607,E2 -13833.607} C_VEL
LIN {X 0,Y 347.791,Z 201.164,A -85,B 0,C 180,E1 -13836.162,E2 -13836.162} C_VEL
LIN {X 0,Y 347.815,Z 201.16,A -85,B 0,C 180,E1 -13839.909,E2 -13839.909} C_VEL
LIN {X 0,Y 347.869,Z 201.153,A -85,B 0,C 180,E1 -13842.359,E2 -13842.359} C_VEL
LIN {X 0,Y 347.9,Z 201.149,A -85,B 0,C 180,E1 -13845.97,E2 -13845.97} C_VEL
LIN {X 0,Y 347.918,Z 201.158,A -85,B 0,C 180,E1 -13850.113,E2 -13850.113} C_VEL
LIN {X 0,Y 347.956,Z 201.366,A -85,B 0,C 180,E1 -13850.407,E2 -13850.407} C_VEL
LIN {X 0,Y 350.205,Z 208.067,A -85,B 0,C 180,E1 -13852.538,E2 -13852.538} C_VEL
LIN {X 0,Y 352.398,Z 216.328,A -85,B 0,C 180,E1 -13854.908,E2 -13854.908} C_VEL
LIN {X 0,Y 354.199,Z 223.56,A -85,B 0,C 180,E1 -13856.872,E2 -13856.872} C_VEL
LIN {X 0,Y 354.064,Z 228.482,A -85,B 0,C 180,E1 -13858.009,E2 -13858.009} C_VEL
LIN {X 0,Y 353.706,Z 233.61,A -85,B 0,C 180,E1 -13859.11,E2 -13859.11} C_VEL
LIN {X 0,Y 357.936,Z 251.285,A -85,B 0,C 180,E1 -13860.151,E2 -13860.151} C_VEL
LIN {X 0,Y 358.876,Z 256.828,A -85,B 0,C 180,E1 -13860.426,E2 -13860.426} C_VEL
LIN {X 0,Y 356.27,Z 319.886,A -85,B 0,C 180,E1 -13862.296,E2 -13862.296} C_VEL
LIN {X 0,Y 355.688,Z 332.423,A -85,B 0,C 180,E1 -13862.902,E2 -13862.902} C_VEL
LIN {X 0,Y 354.899,Z 343.83,A -85,B 0,C 180,E1 -13863.69,E2 -13863.69} C_VEL
LIN {X 0,Y 354.036,Z 353.44,A -85,B 0,C 180,E1 -13864.554,E2 -13864.554} C_VEL
LIN {X 0,Y 353.016,Z 363.503,A -85,B 0,C 180,E1 -13865.712,E2 -13865.712} C_VEL
LIN {X 0,Y 352.025,Z 371.627,A -85,B 0,C 180,E1 -13866.879,E2 -13866.879} C_VEL
LIN {X 0,Y 350.946,Z 379.817,A -85,B 0,C 180,E1 -13868.348,E2 -13868.348} C_VEL
LIN {X 0,Y 349.948,Z 386.571,A -85,B 0,C 180,E1 -13869.882,E2 -13869.882} C_VEL
LIN {X 0,Y 349.03,Z 392.463,A -85,B 0,C 180,E1 -13871.616,E2 -13871.616} C_VEL
LIN {X 0,Y 348.267,Z 396.914,A -85,B 0,C 180,E1 -13873.418,E2 -13873.418} C_VEL
LIN {X 0,Y 347.636,Z 399.985,A -85,B 0,C 180,E1 -13875.237,E2 -13875.237} C_VEL
LIN {X 0,Y 347.329,Z 401.252,A -85,B 0,C 180,E1 -13876.456,E2 -13876.456} C_VEL
LIN {X 0,Y 347.06,Z 402.017,A -85,B 0,C 180,E1 -13877.87,E2 -13877.87} C_VEL
LIN {X 0,Y 346.92,Z 402.108,A -85,B 0,C 180,E1 -13878.912,E2 -13878.912} C_VEL
LIN {X 0,Y 346.805,Z 401.644,A -85,B 0,C 180,E1 -13880.151,E2 -13880.151} C_VEL
LIN {X 0,Y 346.78,Z 400.611,A -85,B 0,C 180,E1 -13881.394,E2 -13881.394} C_VEL
LIN {X 0,Y 346.903,Z 397.876,A -85,B 0,C 180,E1 -13883.269,E2 -13883.269} C_VEL
LIN {X 0,Y 347.161,Z 393.623,A -85,B 0,C 180,E1 -13885.158,E2 -13885.158} C_VEL
LIN {X 0,Y 347.488,Z 388.595,A -85,B 0,C 180,E1 -13886.79,E2 -13886.79} C_VEL
LIN {X 0,Y 347.804,Z 382.411,A -85,B 0,C 180,E1 -13888.349,E2 -13888.349} C_VEL
LIN {X 0,Y 348.394,Z 374.078,A -85,B 0,C 180,E1 -13889.995,E2 -13889.995} C_VEL
LIN {X 0,Y 348.987,Z 364.986,A -85,B 0,C 180,E1 -13891.404,E2 -13891.404} C_VEL
LIN {X 0,Y 349.532,Z 355.904,A -85,B 0,C 180,E1 -13892.528,E2 -13892.528} C_VEL
LIN {X 0,Y 350.083,Z 345.993,A -85,B 0,C 180,E1 -13893.508,E2 -13893.508} C_VEL
LIN {X 0,Y 350.563,Z 334.56,A -85,B 0,C 180,E1 -13894.379,E2 -13894.379} C_VEL
LIN {X 0,Y 350.999,Z 322.569,A -85,B 0,C 180,E1 -13895.039,E2 -13895.039} C_VEL
LIN {X 0,Y 351.144,Z 310.348,A -85,B 0,C 180,E1 -13895.479,E2 -13895.479} C_VEL
LIN {X 0,Y 352.405,Z 250.579,A -85,B 0,C 180,E1 -13897.028,E2 -13897.028} C_VEL
LIN {X 0,Y 349.405,Z 230.613,A -85,B 0,C 180,E1 -13897.716,E2 -13897.716} C_VEL
LIN {X 0,Y 350.124,Z 214.594,A -85,B 0,C 180,E1 -13901.483,E2 -13901.483} C_VEL
LIN {X 0,Y 349.492,Z 209.752,A -85,B 0,C 180,E1 -13902.697,E2 -13902.697} C_VEL
LIN {X 0,Y 347.841,Z 201.4,A -85,B 0,C 180,E1 -13904.893,E2 -13904.893} C_VEL
LIN {X 0,Y 347.749,Z 201.168,A -85,B 0,C 180,E1 -13908.397,E2 -13908.397} C_VEL
LIN {X 0,Y 347.772,Z 201.164,A -85,B 0,C 180,E1 -13912.011,E2 -13912.011} C_VEL
LIN {X 0,Y 347.743,Z 201.171,A -85,B 0,C 180,E1 -13915.535,E2 -13915.535} C_VEL
LIN {X 0,Y 347.763,Z 201.168,A -85,B 0,C 180,E1 -13919.653,E2 -13919.653} C_VEL
LIN {X 0,Y 347.85,Z 201.152,A -85,B 0,C 180,E1 -13922.744,E2 -13922.744} C_VEL
LIN {X 0,Y 347.787,Z 201.16,A -85,B 0,C 180,E1 -13926.161,E2 -13926.161} C_VEL
LIN {X 0,Y 347.816,Z 201.158,A -85,B 0,C 180,E1 -13929.909,E2 -13929.909} C_VEL
LIN {X 0,Y 347.865,Z 201.15,A -85,B 0,C 180,E1 -13932.359,E2 -13932.359} C_VEL
LIN {X 0,Y 347.895,Z 201.147,A -85,B 0,C 180,E1 -13935.97,E2 -13935.97} C_VEL
LIN {X 0,Y 347.927,Z 201.146,A -85,B 0,C 180,E1 -13939.525,E2 -13939.525} C_VEL
LIN {X 0,Y 348.072,Z 201.125,A -85,B 0,C 180,E1 -13941.874,E2 -13941.874} C_VEL
LIN {X 0,Y 348.066,Z 201.125,A -85,B 0,C 180,E1 -13944.205,E2 -13944.205} C_VEL
LIN {X 0,Y 348.205,Z 201.109,A -85,B 0,C 180,E1 -13947.686,E2 -13947.686} C_VEL
LIN {X 0,Y 348.344,Z 201.09,A -85,B 0,C 180,E1 -13949.999,E2 -13949.999} C_VEL
LIN {X 0,Y 348.205,Z 201.108,A -85,B 0,C 180,E1 -13952.313,E2 -13952.313} C_VEL
LIN {X 0,Y 348.088,Z 201.128,A -85,B 0,C 180,E1 -13956.957,E2 -13956.957} C_VEL
LIN {X 0,Y 347.925,Z 201.145,A -85,B 0,C 180,E1 -13960.474,E2 -13960.474} C_VEL
LIN {X 0,Y 347.894,Z 201.147,A -85,B 0,C 180,E1 -13964.149,E2 -13964.149} C_VEL
LIN {X 0,Y 347.887,Z 201.149,A -85,B 0,C 180,E1 -13968.29,E2 -13968.29} C_VEL
LIN {X 0,Y 347.783,Z 201.16,A -85,B 0,C 180,E1 -13971.634,E2 -13971.634} C_VEL
LIN {X 0,Y 347.802,Z 201.159,A -85,B 0,C 180,E1 -13975.203,E2 -13975.203} C_VEL
LIN {X 0,Y 347.805,Z 201.157,A -85,B 0,C 180,E1 -13977.693,E2 -13977.693} C_VEL
LIN {X 0,Y 347.762,Z 201.165,A -85,B 0,C 180,E1 -13980.233,E2 -13980.233} C_VEL
LIN {X 0,Y 347.082,Z 201.256,A -85,B 0,C 180,E1 -13981.198,E2 -13981.198} C_VEL
LIN {X 0,Y 344.255,Z 201.609,A -85,B 0,C 180,E1 -13982.77,E2 -13982.77} C_VEL
LIN {X 0,Y 341.857,Z 201.903,A -85,B 0,C 180,E1 -13984.041,E2 -13984.041} C_VEL
LIN {X 0,Y 340.806,Z 202.032,A -85,B 0,C 180,E1 -13985.025,E2 -13985.025} C_VEL
LIN {X 0,Y 340.708,Z 202.042,A -85,B 0,C 180,E1 -13985.358,E2 -13985.358} C_VEL
LIN {X 0,Y 340.711,Z 202.046,A -85,B 0,C 180,E1 -13988.387,E2 -13988.387} C_VEL
LIN {X 0,Y 340.719,Z 202.04,A -85,B 0,C 180,E1 -13991.303,E2 -13991.303} C_VEL
LIN {X 0,Y 340.73,Z 202.043,A -85,B 0,C 180,E1 -13994.529,E2 -13994.529} C_VEL
LIN {X 0,Y 340.726,Z 202.042,A -85,B 0,C 180,E1 -13997.948,E2 -13997.948} C_VEL
LIN {X 0,Y 340.733,Z 202.04,A -85,B 0,C 180,E1 -14001.773,E2 -14001.773} C_VEL
LIN {X 0,Y 340.715,Z 202.042,A -85,B 0,C 180,E1 -14005.595,E2 -14005.595} C_VEL
LIN {X 0,Y 340.709,Z 202.042,A -85,B 0,C 180,E1 -14008.957,E2 -14008.957} C_VEL
LIN {X 0,Y 340.772,Z 202.036,A -85,B 0,C 180,E1 -14012.474,E2 -14012.474} C_VEL
LIN {X 0,Y 340.748,Z 202.039,A -85,B 0,C 180,E1 -14015.638,E2 -14015.638} C_VEL
LIN {X 0,Y 340.74,Z 202.039,A -85,B 0,C 180,E1 -14019.474,E2 -14019.474} C_VEL
LIN {X 0,Y 340.85,Z 202.03,A -85,B 0,C 180,E1 -14021.984,E2 -14021.984} C_VEL
LIN {X 0,Y 340.861,Z 202.027,A -85,B 0,C 180,E1 -14025.705,E2 -14025.705} C_VEL
LIN {X 0,Y 340.863,Z 202.024,A -85,B 0,C 180,E1 -14029.307,E2 -14029.307} C_VEL
LIN {X 0,Y 341.051,Z 201.999,A -85,B 0,C 180,E1 -14032.898,E2 -14032.898} C_VEL
LIN {X 0,Y 341.16,Z 201.991,A -85,B 0,C 180,E1 -14037.639,E2 -14037.639} C_VEL
LIN {X 0,Y 341.288,Z 201.972,A -85,B 0,C 180,E1 -14040.001,E2 -14040.001} C_VEL
LIN {X 0,Y 341.16,Z 201.986,A -85,B 0,C 180,E1 -14042.362,E2 -14042.362} C_VEL
LIN {X 0,Y 341.067,Z 201.999,A -85,B 0,C 180,E1 -14047.103,E2 -14047.103} C_VEL
LIN {X 0,Y 340.864,Z 202.022,A -85,B 0,C 180,E1 -14050.695,E2 -14050.695} C_VEL
LIN {X 0,Y 340.856,Z 202.023,A -85,B 0,C 180,E1 -14054.326,E2 -14054.326} C_VEL
LIN {X 0,Y 340.831,Z 202.026,A -85,B 0,C 180,E1 -14058.467,E2 -14058.467} C_VEL
LIN {X 0,Y 340.748,Z 202.038,A -85,B 0,C 180,E1 -14061.858,E2 -14061.858} C_VEL
LIN {X 0,Y 340.767,Z 202.037,A -85,B 0,C 180,E1 -14065.665,E2 -14065.665} C_VEL
LIN {X 0,Y 340.723,Z 202.04,A -85,B 0,C 180,E1 -14068.322,E2 -14068.322} C_VEL
LIN {X 0,Y 340.693,Z 202.048,A -85,B 0,C 180,E1 -14071.046,E2 -14071.046} C_VEL
LIN {X 0,Y 340.713,Z 202.045,A -85,B 0,C 180,E1 -14075.28,E2 -14075.28} C_VEL
LIN {X 0,Y 340.705,Z 202.043,A -85,B 0,C 180,E1 -14078.387,E2 -14078.387} C_VEL
LIN {X 0,Y 340.695,Z 202.043,A -85,B 0,C 180,E1 -14082.047,E2 -14082.047} C_VEL
LIN {X 0,Y 340.649,Z 202.049,A -85,B 0,C 180,E1 -14086.228,E2 -14086.228} C_VEL
LIN {X 0,Y 340.685,Z 202.045,A -85,B 0,C 180,E1 -14089.754,E2 -14089.754} C_VEL
LIN {X 0,Y 340.703,Z 202.048,A -85,B 0,C 180,E1 -14093.26,E2 -14093.26} C_VEL
LIN {X 0,Y 340.711,Z 202.047,A -85,B 0,C 180,E1 -14096.865,E2 -14096.865} C_VEL
LIN {X 0,Y 340.782,Z 202.337,A -85,B 0,C 180,E1 -14097.445,E2 -14097.445} C_VEL
LIN {X 0,Y 344.527,Z 218.694,A -85,B 0,C 180,E1 -14100.935,E2 -14100.935} C_VEL
LIN {X 0,Y 346.367,Z 227.938,A -85,B 0,C 180,E1 -14102.818,E2 -14102.818} C_VEL
LIN {X 0,Y 344.641,Z 244.787,A -85,B 0,C 180,E1 -14105.932,E2 -14105.932} C_VEL
LIN {X 0,Y 343.175,Z 260.593,A -85,B 0,C 180,E1 -14108.782,E2 -14108.782} C_VEL
LIN {X 0,Y 346.107,Z 294.639,A -85,B 0,C 180,E1 -14109.772,E2 -14109.772} C_VEL
LIN {X 0,Y 344.792,Z 366.231,A -85,B 0,C 180,E1 -14111.506,E2 -14111.506} C_VEL
LIN {X 0,Y 344.134,Z 379.169,A -85,B 0,C 180,E1 -14112.047,E2 -14112.047} C_VEL
LIN {X 0,Y 343.432,Z 390.597,A -85,B 0,C 180,E1 -14112.74,E2 -14112.74} C_VEL
LIN {X 0,Y 342.595,Z 403.135,A -85,B 0,C 180,E1 -14113.77,E2 -14113.77} C_VEL
LIN {X 0,Y 341.736,Z 414.392,A -85,B 0,C 180,E1 -14114.965,E2 -14114.965} C_VEL
LIN {X 0,Y 341.01,Z 424.288,A -85,B 0,C 180,E1 -14116.291,E2 -14116.291} C_VEL
LIN {X 0,Y 340.273,Z 433.308,A -85,B 0,C 180,E1 -14117.779,E2 -14117.779} C_VEL
LIN {X 0,Y 339.815,Z 440.714,A -85,B 0,C 180,E1 -14119.274,E2 -14119.274} C_VEL
LIN {X 0,Y 339.538,Z 447.887,A -85,B 0,C 180,E1 -14121.07,E2 -14121.07} C_VEL
LIN {X 0,Y 339.535,Z 453.547,A -85,B 0,C 180,E1 -14122.867,E2 -14122.867} C_VEL
LIN {X 0,Y 339.526,Z 457.879,A -85,B 0,C 180,E1 -14124.656,E2 -14124.656} C_VEL
LIN {X 0,Y 339.636,Z 461.034,A -85,B 0,C 180,E1 -14126.442,E2 -14126.442} C_VEL
LIN {X 0,Y 339.762,Z 462.552,A -85,B 0,C 180,E1 -14127.63,E2 -14127.63} C_VEL
LIN {X 0,Y 339.718,Z 463.544,A -85,B 0,C 180,E1 -14128.815,E2 -14128.815} C_VEL
LIN {X 0,Y 339.685,Z 464.103,A -85,B 0,C 180,E1 -14130.001,E2 -14130.001} C_VEL
LIN {X 0,Y 339.703,Z 464.24,A -85,B 0,C 180,E1 -14131.186,E2 -14131.186} C_VEL
LIN {X 0,Y 339.594,Z 463.884,A -85,B 0,C 180,E1 -14132.373,E2 -14132.373} C_VEL
LIN {X 0,Y 339.445,Z 463.089,A -85,B 0,C 180,E1 -14133.562,E2 -14133.562} C_VEL
LIN {X 0,Y 339.377,Z 461.883,A -85,B 0,C 180,E1 -14134.752,E2 -14134.752} C_VEL
LIN {X 0,Y 339.357,Z 459.718,A -85,B 0,C 180,E1 -14136.24,E2 -14136.24} C_VEL
LIN {X 0,Y 339.421,Z 455.484,A -85,B 0,C 180,E1 -14138.335,E2 -14138.335} C_VEL
LIN {X 0,Y 339.675,Z 450.614,A -85,B 0,C 180,E1 -14140.13,E2 -14140.13} C_VEL
LIN {X 0,Y 340.341,Z 444.448,A -85,B 0,C 180,E1 -14141.918,E2 -14141.918} C_VEL
LIN {X 0,Y 341.188,Z 436.768,A -85,B 0,C 180,E1 -14143.703,E2 -14143.703} C_VEL
LIN {X 0,Y 342.332,Z 428.266,A -85,B 0,C 180,E1 -14145.302,E2 -14145.302} C_VEL
LIN {X 0,Y 343.627,Z 418.5,A -85,B 0,C 180,E1 -14146.792,E2 -14146.792} C_VEL
LIN {X 0,Y 345.195,Z 407.845,A -85,B 0,C 180,E1 -14148.089,E2 -14148.089} C_VEL
LIN {X 0,Y 346.649,Z 395.941,A -85,B 0,C 180,E1 -14149.236,E2 -14149.236} C_VEL
LIN {X 0,Y 348.066,Z 383.31,A -85,B 0,C 180,E1 -14150.153,E2 -14150.153} C_VEL
LIN {X 0,Y 349.217,Z 370.637,A -85,B 0,C 180,E1 -14150.814,E2 -14150.814} C_VEL
LIN {X 0,Y 349.957,Z 357.551,A -85,B 0,C 180,E1 -14151.266,E2 -14151.266} C_VEL
LIN {X 0,Y 351.981,Z 294.385,A -85,B 0,C 180,E1 -14152.891,E2 -14152.891} C_VEL
LIN {X 0,Y 350.067,Z 275.45,A -85,B 0,C 180,E1 -14153.641,E2 -14153.641} C_VEL
LIN {X 0,Y 347.178,Z 258.191,A -85,B 0,C 180,E1 -14154.469,E2 -14154.469} C_VEL
LIN {X 0,Y 347.058,Z 257.135,A -85,B 0,C 180,E1 -14154.549,E2 -14154.549} C_VEL
LIN {X 0,Y 349.743,Z 237.185,A -85,B 0,C 180,E1 -14158.179,E2 -14158.179} C_VEL
LIN {X 0,Y 349.949,Z 235.53,A -85,B 0,C 180,E1 -14158.488,E2 -14158.488} C_VEL
LIN {X 0,Y 348.172,Z 226.398,A -85,B 0,C 180,E1 -14160.593,E2 -14160.593} C_VEL
LIN {X 0,Y 345.204,Z 215.389,A -85,B 0,C 180,E1 -14163.413,E2 -14163.413} C_VEL
LIN {X 0,Y 342.833,Z 208.216,A -85,B 0,C 180,E1 -14165.469,E2 -14165.469} C_VEL
LIN {X 0,Y 340.737,Z 202.146,A -85,B 0,C 180,E1 -14167.444,E2 -14167.444} C_VEL
LIN {X 0,Y 340.674,Z 202.049,A -85,B 0,C 180,E1 -14171.312,E2 -14171.312} C_VEL
LIN {X 0,Y 340.644,Z 202.051,A -85,B 0,C 180,E1 -14174.546,E2 -14174.546} C_VEL
LIN {X 0,Y 340.702,Z 202.042,A -85,B 0,C 180,E1 -14177.955,E2 -14177.955} C_VEL
LIN {X 0,Y 340.736,Z 202.039,A -85,B 0,C 180,E1 -14181.772,E2 -14181.772} C_VEL
LIN {X 0,Y 340.726,Z 202.042,A -85,B 0,C 180,E1 -14185.595,E2 -14185.595} C_VEL
LIN {X 0,Y 340.701,Z 202.043,A -85,B 0,C 180,E1 -14188.955,E2 -14188.955} C_VEL
LIN {X 0,Y 340.806,Z 202.03,A -85,B 0,C 180,E1 -14193.02,E2 -14193.02} C_VEL
LIN {X 0,Y 340.732,Z 202.039,A -85,B 0,C 180,E1 -14196.927,E2 -14196.927} C_VEL
LIN {X 0,Y 340.794,Z 202.033,A -85,B 0,C 180,E1 -14200.733,E2 -14200.733} C_VEL
LIN {X 0,Y 340.789,Z 202.035,A -85,B 0,C 180,E1 -14203.218,E2 -14203.218} C_VEL
LIN {X 0,Y 340.847,Z 202.029,A -85,B 0,C 180,E1 -14206.89,E2 -14206.89} C_VEL
LIN {X 0,Y 340.888,Z 202.202,A -85,B 0,C 180,E1 -14209.344,E2 -14209.344} C_VEL
LIN {X 0,Y 343.937,Z 211.247,A -85,B 0,C 180,E1 -14212.367,E2 -14212.367} C_VEL
LIN {X 0,Y 346.343,Z 220.543,A -85,B 0,C 180,E1 -14215.095,E2 -14215.095} C_VEL
LIN {X 0,Y 347.771,Z 226.75,A -85,B 0,C 180,E1 -14216.814,E2 -14216.814} C_VEL
LIN {X 0,Y 347.271,Z 234.012,A -85,B 0,C 180,E1 -14218.441,E2 -14218.441} C_VEL
LIN {X 0,Y 351.414,Z 250.796,A -85,B 0,C 180,E1 -14219.502,E2 -14219.502} C_VEL
LIN {X 0,Y 352.717,Z 257.71,A -85,B 0,C 180,E1 -14219.868,E2 -14219.868} C_VEL
LIN {X 0,Y 349.952,Z 319.768,A -85,B 0,C 180,E1 -14221.762,E2 -14221.762} C_VEL
LIN {X 0,Y 349.348,Z 332.401,A -85,B 0,C 180,E1 -14222.377,E2 -14222.377} C_VEL
LIN {X 0,Y 348.504,Z 343.977,A -85,B 0,C 180,E1 -14223.179,E2 -14223.179} C_VEL
LIN {X 0,Y 347.449,Z 355.099,A -85,B 0,C 180,E1 -14224.204,E2 -14224.204} C_VEL
LIN {X 0,Y 346.351,Z 365.098,A -85,B 0,C 180,E1 -14225.397,E2 -14225.397} C_VEL
LIN {X 0,Y 345.194,Z 373.857,A -85,B 0,C 180,E1 -14226.722,E2 -14226.722} C_VEL
LIN {X 0,Y 344.061,Z 381.727,A -85,B 0,C 180,E1 -14228.22,E2 -14228.22} C_VEL
LIN {X 0,Y 342.916,Z 388.911,A -85,B 0,C 180,E1 -14229.978,E2 -14229.978} C_VEL
LIN {X 0,Y 341.894,Z 394.657,A -85,B 0,C 180,E1 -14231.862,E2 -14231.862} C_VEL
LIN {X 0,Y 341.132,Z 398.689,A -85,B 0,C 180,E1 -14233.704,E2 -14233.704} C_VEL
LIN {X 0,Y 340.515,Z 401.329,A -85,B 0,C 180,E1 -14235.563,E2 -14235.563} C_VEL
LIN {X 0,Y 340.189,Z 402.352,A -85,B 0,C 180,E1 -14236.811,E2 -14236.811} C_VEL
LIN {X 0,Y 339.994,Z 402.812,A -85,B 0,C 180,E1 -14238.062,E2 -14238.062} C_VEL
LIN {X 0,Y 339.801,Z 402.666,A -85,B 0,C 180,E1 -14239.324,E2 -14239.324} C_VEL
LIN {X 0,Y 339.721,Z 401.155,A -85,B 0,C 180,E1 -14241.417,E2 -14241.417} C_VEL
LIN {X 0,Y 339.809,Z 398.681,A -85,B 0,C 180,E1 -14243.138,E2 -14243.138} C_VEL
LIN {X 0,Y 340.077,Z 394.469,A -85,B 0,C 180,E1 -14245.076,E2 -14245.076} C_VEL
LIN {X 0,Y 340.452,Z 388.563,A -85,B 0,C 180,E1 -14247.009,E2 -14247.009} C_VEL
LIN {X 0,Y 340.81,Z 381.955,A -85,B 0,C 180,E1 -14248.649,E2 -14248.649} C_VEL
LIN {X 0,Y 341.381,Z 374.283,A -85,B 0,C 180,E1 -14250.156,E2 -14250.156} C_VEL
LIN {X 0,Y 342.005,Z 365.038,A -85,B 0,C 180,E1 -14251.601,E2 -14251.601} C_VEL
LIN {X 0,Y 342.612,Z 354.94,A -85,B 0,C 180,E1 -14252.842,E2 -14252.842} C_VEL
LIN {X 0,Y 343.23,Z 343.735,A -85,B 0,C 180,E1 -14253.915,E2 -14253.915} C_VEL
LIN {X 0,Y 343.702,Z 332.226,A -85,B 0,C 180,E1 -14254.749,E2 -14254.749} C_VEL
LIN {X 0,Y 344.044,Z 319.85,A -85,B 0,C 180,E1 -14255.382,E2 -14255.382} C_VEL
LIN {X 0,Y 344.35,Z 304.516,A -85,B 0,C 180,E1 -14255.854,E2 -14255.854} C_VEL
LIN {X 0,Y 345.503,Z 251.486,A -85,B 0,C 180,E1 -14257.264,E2 -14257.264} C_VEL
LIN {X 0,Y 342.443,Z 231.108,A -85,B 0,C 180,E1 -14257.973,E2 -14257.973} C_VEL
LIN {X 0,Y 343.104,Z 216.812,A -85,B 0,C 180,E1 -14261.345,E2 -14261.345} C_VEL
LIN {X 0,Y 342.788,Z 212.473,A -85,B 0,C 180,E1 -14262.431,E2 -14262.431} C_VEL
LIN {X 0,Y 340.75,Z 202.18,A -85,B 0,C 180,E1 -14265.193,E2 -14265.193} C_VEL
LIN {X 0,Y 340.684,Z 202.047,A -85,B 0,C 180,E1 -14268.69,E2 -14268.69} C_VEL
LIN {X 0,Y 340.731,Z 202.044,A -85,B 0,C 180,E1 -14271.772,E2 -14271.772} C_VEL
LIN {X 0,Y 340.722,Z 202.046,A -85,B 0,C 180,E1 -14275.595,E2 -14275.595} C_VEL
LIN {X 0,Y 340.703,Z 202.043,A -85,B 0,C 180,E1 -14278.955,E2 -14278.955} C_VEL
LIN {X 0,Y 340.777,Z 202.033,A -85,B 0,C 180,E1 -14282.473,E2 -14282.473} C_VEL
LIN {X 0,Y 340.755,Z 202.04,A -85,B 0,C 180,E1 -14285.638,E2 -14285.638} C_VEL
LIN {X 0,Y 340.747,Z 202.042,A -85,B 0,C 180,E1 -14289.474,E2 -14289.474} C_VEL
LIN {X 0,Y 340.856,Z 202.024,A -85,B 0,C 180,E1 -14291.983,E2 -14291.983} C_VEL
LIN {X 0,Y 340.867,Z 202.024,A -85,B 0,C 180,E1 -14295.704,E2 -14295.704} C_VEL
LIN {X 0,Y 340.869,Z 202.027,A -85,B 0,C 180,E1 -14299.305,E2 -14299.305} C_VEL
LIN {X 0,Y 341.074,Z 201.999,A -85,B 0,C 180,E1 -14302.897,E2 -14302.897} C_VEL
LIN {X 0,Y 341.167,Z 201.986,A -85,B 0,C 180,E1 -14307.638,E2 -14307.638} C_VEL
LIN {X 0,Y 341.294,Z 201.969,A -85,B 0,C 180,E1 -14309.999,E2 -14309.999} C_VEL
LIN {X 0,Y 341.167,Z 201.985,A -85,B 0,C 180,E1 -14312.36,E2 -14312.36} C_VEL
LIN {X 0,Y 341.056,Z 202.003,A -85,B 0,C 180,E1 -14317.101,E2 -14317.101} C_VEL
LIN {X 0,Y 340.867,Z 202.026,A -85,B 0,C 180,E1 -14320.693,E2 -14320.693} C_VEL
LIN {X 0,Y 340.858,Z 202.024,A -85,B 0,C 180,E1 -14324.324,E2 -14324.324} C_VEL
LIN {X 0,Y 340.833,Z 202.029,A -85,B 0,C 180,E1 -14328.466,E2 -14328.466} C_VEL
LIN {X 0,Y 340.748,Z 202.037,A -85,B 0,C 180,E1 -14331.856,E2 -14331.856} C_VEL
LIN {X 0,Y 340.767,Z 202.034,A -85,B 0,C 180,E1 -14335.664,E2 -14335.664} C_VEL
LIN {X 0,Y 340.735,Z 202.041,A -85,B 0,C 180,E1 -14338.319,E2 -14338.319} C_VEL
LIN {X 0,Y 340.697,Z 202.045,A -85,B 0,C 180,E1 -14341.043,E2 -14341.043} C_VEL
LIN {X 0,Y 340.713,Z 202.041,A -85,B 0,C 180,E1 -14345.278,E2 -14345.278} C_VEL
LIN {X 0,Y 340.708,Z 202.042,A -85,B 0,C 180,E1 -14345.358,E2 -14345.358} C_VEL
LIN {X 0,Y 339.999,Z 202.134,A -85,B 0,C 180,E1 -14346.345,E2 -14346.345} C_VEL
LIN {X 0,Y 337.114,Z 202.491,A -85,B 0,C 180,E1 -14347.951,E2 -14347.951} C_VEL
LIN {X 0,Y 334.723,Z 202.787,A -85,B 0,C 180,E1 -14349.252,E2 -14349.252} C_VEL
LIN {X 0,Y 333.743,Z 202.913,A -85,B 0,C 180,E1 -14350.259,E2 -14350.259} C_VEL
LIN {X 0,Y 333.687,Z 202.919,A -85,B 0,C 180,E1 -14350.6,E2 -14350.6} C_VEL
LIN {X 0,Y 333.672,Z 202.923,A -85,B 0,C 180,E1 -14354.265,E2 -14354.265} C_VEL
LIN {X 0,Y 333.674,Z 202.918,A -85,B 0,C 180,E1 -14357.624,E2 -14357.624} C_VEL
LIN {X 0,Y 333.67,Z 202.918,A -85,B 0,C 180,E1 -14361.196,E2 -14361.196} C_VEL
LIN {X 0,Y 333.677,Z 202.917,A -85,B 0,C 180,E1 -14365.226,E2 -14365.226} C_VEL
LIN {X 0,Y 333.638,Z 202.928,A -85,B 0,C 180,E1 -14368.223,E2 -14368.223} C_VEL
LIN {X 0,Y 333.704,Z 202.914,A -85,B 0,C 180,E1 -14371.028,E2 -14371.028} C_VEL
LIN {X 0,Y 333.728,Z 202.914,A -85,B 0,C 180,E1 -14373.754,E2 -14373.754} C_VEL
LIN {X 0,Y 333.711,Z 202.918,A -85,B 0,C 180,E1 -14377.914,E2 -14377.914} C_VEL
LIN {X 0,Y 333.786,Z 202.906,A -85,B 0,C 180,E1 -14381.59,E2 -14381.59} C_VEL
LIN {X 0,Y 333.8,Z 202.905,A -85,B 0,C 180,E1 -14385.577,E2 -14385.577} C_VEL
LIN {X 0,Y 333.826,Z 202.899,A -85,B 0,C 180,E1 -14389.078,E2 -14389.078} C_VEL
LIN {X 0,Y 333.998,Z 202.877,A -85,B 0,C 180,E1 -14392.748,E2 -14392.748} C_VEL
LIN {X 0,Y 333.801,Z 202.903,A -85,B 0,C 180,E1 -14395.17,E2 -14395.17} C_VEL
LIN {X 0,Y 334.097,Z 202.87,A -85,B 0,C 180,E1 -14397.589,E2 -14397.589} C_VEL
LIN {X 0,Y 334.239,Z 202.85,A -85,B 0,C 180,E1 -14400.001,E2 -14400.001} C_VEL
LIN {X 0,Y 334.098,Z 202.865,A -85,B 0,C 180,E1 -14402.412,E2 -14402.412} C_VEL
LIN {X 0,Y 334.017,Z 202.878,A -85,B 0,C 180,E1 -14407.253,E2 -14407.253} C_VEL
LIN {X 0,Y 333.827,Z 202.9,A -85,B 0,C 180,E1 -14410.923,E2 -14410.923} C_VEL
LIN {X 0,Y 333.802,Z 202.902,A -85,B 0,C 180,E1 -14414.635,E2 -14414.635} C_VEL
LIN {X 0,Y 333.79,Z 202.904,A -85,B 0,C 180,E1 -14418.656,E2 -14418.656} C_VEL
LIN {X 0,Y 333.687,Z 202.916,A -85,B 0,C 180,E1 -14422.279,E2 -14422.279} C_VEL
LIN {X 0,Y 333.729,Z 202.911,A -85,B 0,C 180,E1 -14426.247,E2 -14426.247} C_VEL
LIN {X 0,Y 333.685,Z 202.92,A -85,B 0,C 180,E1 -14428.975,E2 -14428.975} C_VEL
LIN {X 0,Y 333.639,Z 202.923,A -85,B 0,C 180,E1 -14432.588,E2 -14432.588} C_VEL
LIN {X 0,Y 333.671,Z 202.918,A -85,B 0,C 180,E1 -14436.14,E2 -14436.14} C_VEL
LIN {X 0,Y 333.642,Z 202.926,A -85,B 0,C 180,E1 -14439.194,E2 -14439.194} C_VEL
LIN {X 0,Y 333.629,Z 202.925,A -85,B 0,C 180,E1 -14442.501,E2 -14442.501} C_VEL
LIN {X 0,Y 333.593,Z 202.928,A -85,B 0,C 180,E1 -14445.956,E2 -14445.956} C_VEL
LIN {X 0,Y 333.644,Z 202.924,A -85,B 0,C 180,E1 -14449.317,E2 -14449.317} C_VEL
LIN {X 0,Y 333.663,Z 202.924,A -85,B 0,C 180,E1 -14453.169,E2 -14453.169} C_VEL
LIN {X 0,Y 333.696,Z 202.972,A -85,B 0,C 180,E1 -14456.975,E2 -14456.975} C_VEL
LIN {X 0,Y 333.755,Z 203.381,A -85,B 0,C 180,E1 -14457.157,E2 -14457.157} C_VEL
LIN {X 0,Y 337.312,Z 218.902,A -85,B 0,C 180,E1 -14460.545,E2 -14460.545} C_VEL
LIN {X 0,Y 339.364,Z 228.563,A -85,B 0,C 180,E1 -14462.564,E2 -14462.564} C_VEL
LIN {X 0,Y 338.601,Z 236.974,A -85,B 0,C 180,E1 -14464.16,E2 -14464.16} C_VEL
LIN {X 0,Y 336.223,Z 260.098,A -85,B 0,C 180,E1 -14468.476,E2 -14468.476} C_VEL
LIN {X 0,Y 339.175,Z 295.436,A -85,B 0,C 180,E1 -14469.536,E2 -14469.536} C_VEL
LIN {X 0,Y 337.845,Z 365.431,A -85,B 0,C 180,E1 -14471.269,E2 -14471.269} C_VEL
LIN {X 0,Y 337.178,Z 378.438,A -85,B 0,C 180,E1 -14471.821,E2 -14471.821} C_VEL
LIN {X 0,Y 336.455,Z 389.917,A -85,B 0,C 180,E1 -14472.527,E2 -14472.527} C_VEL
LIN {X 0,Y 335.603,Z 402.481,A -85,B 0,C 180,E1 -14473.579,E2 -14473.579} C_VEL
LIN {X 0,Y 334.797,Z 412.765,A -85,B 0,C 180,E1 -14474.68,E2 -14474.68} C_VEL
LIN {X 0,Y 333.973,Z 422.65,A -85,B 0,C 180,E1 -14475.996,E2 -14475.996} C_VEL
LIN {X 0,Y 333.271,Z 431.854,A -85,B 0,C 180,E1 -14477.518,E2 -14477.518} C_VEL
LIN {X 0,Y 332.795,Z 439.404,A -85,B 0,C 180,E1 -14479.045,E2 -14479.045} C_VEL
LIN {X 0,Y 332.482,Z 446.749,A -85,B 0,C 180,E1 -14480.879,E2 -14480.879} C_VEL
LIN {X 0,Y 332.447,Z 452.507,A -85,B 0,C 180,E1 -14482.714,E2 -14482.714} C_VEL
LIN {X 0,Y 332.476,Z 456.935,A -85,B 0,C 180,E1 -14484.543,E2 -14484.543} C_VEL
LIN {X 0,Y 332.576,Z 460.17,A -85,B 0,C 180,E1 -14486.366,E2 -14486.366} C_VEL
LIN {X 0,Y 332.7,Z 461.732,A -85,B 0,C 180,E1 -14487.58,E2 -14487.58} C_VEL
LIN {X 0,Y 332.674,Z 462.787,A -85,B 0,C 180,E1 -14488.79,E2 -14488.79} C_VEL
LIN {X 0,Y 332.639,Z 463.375,A -85,B 0,C 180,E1 -14490.001,E2 -14490.001} C_VEL
LIN {X 0,Y 332.655,Z 463.544,A -85,B 0,C 180,E1 -14491.211,E2 -14491.211} C_VEL
LIN {X 0,Y 332.524,Z 463.248,A -85,B 0,C 180,E1 -14492.423,E2 -14492.423} C_VEL
LIN {X 0,Y 332.353,Z 462.486,A -85,B 0,C 180,E1 -14493.638,E2 -14493.638} C_VEL
LIN {X 0,Y 332.306,Z 461.315,A -85,B 0,C 180,E1 -14494.854,E2 -14494.854} C_VEL
LIN {X 0,Y 332.262,Z 459.498,A -85,B 0,C 180,E1 -14496.2,E2 -14496.2} C_VEL
LIN {X 0,Y 332.324,Z 456.403,A -85,B 0,C 180,E1 -14497.902,E2 -14497.902} C_VEL
LIN {X 0,Y 332.504,Z 451.98,A -85,B 0,C 180,E1 -14499.736,E2 -14499.736} C_VEL
LIN {X 0,Y 333.196,Z 445.268,A -85,B 0,C 180,E1 -14501.869,E2 -14501.869} C_VEL
LIN {X 0,Y 334.075,Z 438.032,A -85,B 0,C 180,E1 -14503.691,E2 -14503.691} C_VEL
LIN {X 0,Y 335.237,Z 429.855,A -85,B 0,C 180,E1 -14505.342,E2 -14505.342} C_VEL
LIN {X 0,Y 336.689,Z 419.741,A -85,B 0,C 180,E1 -14506.992,E2 -14506.992} C_VEL
LIN {X 0,Y 338.259,Z 409.524,A -85,B 0,C 180,E1 -14508.316,E2 -14508.316} C_VEL
LIN {X 0,Y 339.775,Z 398.22,A -85,B 0,C 180,E1 -14509.484,E2 -14509.484} C_VEL
LIN {X 0,Y 341.203,Z 386.571,A -85,B 0,C 180,E1 -14510.419,E2 -14510.419} C_VEL
LIN {X 0,Y 342.638,Z 373.279,A -85,B 0,C 180,E1 -14511.194,E2 -14511.194} C_VEL
LIN {X 0,Y 343.502,Z 360.077,A -85,B 0,C 180,E1 -14511.728,E2 -14511.728} C_VEL
LIN {X 0,Y 345.773,Z 294.358,A -85,B 0,C 180,E1 -14513.477,E2 -14513.477} C_VEL
LIN {X 0,Y 343.805,Z 275.584,A -85,B 0,C 180,E1 -14514.26,E2 -14514.26} C_VEL
LIN {X 0,Y 341.047,Z 259.04,A -85,B 0,C 180,E1 -14515.093,E2 -14515.093} C_VEL
LIN {X 0,Y 340.715,Z 256.592,A -85,B 0,C 180,E1 -14515.262,E2 -14515.262} C_VEL
LIN {X 0,Y 343.413,Z 237.966,A -85,B 0,C 180,E1 -14518.746,E2 -14518.746} C_VEL
LIN {X 0,Y 341.923,Z 229.802,A -85,B 0,C 180,E1 -14520.664,E2 -14520.664} C_VEL
LIN {X 0,Y 339.185,Z 219.301,A -85,B 0,C 180,E1 -14523.417,E2 -14523.417} C_VEL
LIN {X 0,Y 336.631,Z 211.326,A -85,B 0,C 180,E1 -14525.773,E2 -14525.773} C_VEL
LIN {X 0,Y 333.756,Z 203.492,A -85,B 0,C 180,E1 -14528.403,E2 -14528.403} C_VEL
LIN {X 0,Y 333.638,Z 202.956,A -85,B 0,C 180,E1 -14528.794,E2 -14528.794} C_VEL
LIN {X 0,Y 333.632,Z 202.925,A -85,B 0,C 180,E1 -14532.499,E2 -14532.499} C_VEL
LIN {X 0,Y 333.599,Z 202.928,A -85,B 0,C 180,E1 -14535.955,E2 -14535.955} C_VEL
LIN {X 0,Y 333.651,Z 202.923,A -85,B 0,C 180,E1 -14539.315,E2 -14539.315} C_VEL
LIN {X 0,Y 333.668,Z 202.924,A -85,B 0,C 180,E1 -14543.168,E2 -14543.168} C_VEL
LIN {X 0,Y 333.677,Z 202.922,A -85,B 0,C 180,E1 -14545.341,E2 -14545.341} C_VEL
LIN {X 0,Y 333.694,Z 202.919,A -85,B 0,C 180,E1 -14549.637,E2 -14549.637} C_VEL
LIN {X 0,Y 333.743,Z 202.912,A -85,B 0,C 180,E1 -14552.401,E2 -14552.401} C_VEL
LIN {X 0,Y 333.73,Z 202.911,A -85,B 0,C 180,E1 -14555.09,E2 -14555.09} C_VEL
LIN {X 0,Y 333.683,Z 202.918,A -85,B 0,C 180,E1 -14559.019,E2 -14559.019} C_VEL
LIN {X 0,Y 333.797,Z 202.906,A -85,B 0,C 180,E1 -14561.589,E2 -14561.589} C_VEL
LIN {X 0,Y 333.811,Z 202.905,A -85,B 0,C 180,E1 -14565.576,E2 -14565.576} C_VEL
LIN {X 0,Y 333.857,Z 203.106,A -85,B 0,C 180,E1 -14568.194,E2 -14568.194} C_VEL
LIN {X 0,Y 337.192,Z 212.647,A -85,B 0,C 180,E1 -14571.61,E2 -14571.61} C_VEL
LIN {X 0,Y 339.287,Z 220.54,A -85,B 0,C 180,E1 -14574.055,E2 -14574.055} C_VEL
LIN {X 0,Y 341.262,Z 228.877,A -85,B 0,C 180,E1 -14576.457,E2 -14576.457} C_VEL
LIN {X 0,Y 340.95,Z 234.496,A -85,B 0,C 180,E1 -14577.748,E2 -14577.748} C_VEL
LIN {X 0,Y 344.463,Z 248.44,A -85,B 0,C 180,E1 -14578.692,E2 -14578.692} C_VEL
LIN {X 0,Y 346.543,Z 258.558,A -85,B 0,C 180,E1 -14579.285,E2 -14579.285} C_VEL
LIN {X 0,Y 343.669,Z 320.955,A -85,B 0,C 180,E1 -14581.244,E2 -14581.244} C_VEL
LIN {X 0,Y 343.063,Z 332.754,A -85,B 0,C 180,E1 -14581.834,E2 -14581.834} C_VEL
LIN {X 0,Y 342.149,Z 344.345,A -85,B 0,C 180,E1 -14582.648,E2 -14582.648} C_VEL
LIN {X 0,Y 341.015,Z 355.484,A -85,B 0,C 180,E1 -14583.692,E2 -14583.692} C_VEL
LIN {X 0,Y 339.819,Z 365.691,A -85,B 0,C 180,E1 -14584.935,E2 -14584.935} C_VEL
LIN {X 0,Y 338.613,Z 374.31,A -85,B 0,C 180,E1 -14586.255,E2 -14586.255} C_VEL
LIN {X 0,Y 337.414,Z 382.244,A -85,B 0,C 180,E1 -14587.78,E2 -14587.78} C_VEL
LIN {X 0,Y 336.113,Z 389.687,A -85,B 0,C 180,E1 -14589.629,E2 -14589.629} C_VEL
LIN {X 0,Y 335.07,Z 395.257,A -85,B 0,C 180,E1 -14591.493,E2 -14591.493} C_VEL
LIN {X 0,Y 334.218,Z 399.317,A -85,B 0,C 180,E1 -14593.374,E2 -14593.374} C_VEL
LIN {X 0,Y 333.781,Z 401.235,A -85,B 0,C 180,E1 -14594.635,E2 -14594.635} C_VEL
LIN {X 0,Y 333.386,Z 402.563,A -85,B 0,C 180,E1 -14595.905,E2 -14595.905} C_VEL
LIN {X 0,Y 333.068,Z 403.344,A -85,B 0,C 180,E1 -14597.182,E2 -14597.182} C_VEL
LIN {X 0,Y 332.878,Z 403.511,A -85,B 0,C 180,E1 -14598.462,E2 -14598.462} C_VEL
LIN {X 0,Y 332.69,Z 403.112,A -85,B 0,C 180,E1 -14599.754,E2 -14599.754} C_VEL
LIN {X 0,Y 332.646,Z 401.484,A -85,B 0,C 180,E1 -14601.625,E2 -14601.625} C_VEL
LIN {X 0,Y 332.778,Z 398.261,A -85,B 0,C 180,E1 -14603.657,E2 -14603.657} C_VEL
LIN {X 0,Y 333.092,Z 393.58,A -85,B 0,C 180,E1 -14605.628,E2 -14605.628} C_VEL
LIN {X 0,Y 333.439,Z 388.255,A -85,B 0,C 180,E1 -14607.285,E2 -14607.285} C_VEL
LIN {X 0,Y 333.841,Z 381.423,A -85,B 0,C 180,E1 -14608.959,E2 -14608.959} C_VEL
LIN {X 0,Y 334.504,Z 372.423,A -85,B 0,C 180,E1 -14610.673,E2 -14610.673} C_VEL
LIN {X 0,Y 335.175,Z 362.509,A -85,B 0,C 180,E1 -14612.144,E2 -14612.144} C_VEL
LIN {X 0,Y 335.754,Z 352.767,A -85,B 0,C 180,E1 -14613.288,E2 -14613.288} C_VEL
LIN {X 0,Y 336.4,Z 341.294,A -85,B 0,C 180,E1 -14614.338,E2 -14614.338} C_VEL
LIN {X 0,Y 336.871,Z 330.121,A -85,B 0,C 180,E1 -14615.101,E2 -14615.101} C_VEL
LIN {X 0,Y 337.127,Z 318.145,A -85,B 0,C 180,E1 -14615.68,E2 -14615.68} C_VEL
LIN {X 0,Y 337.678,Z 292.134,A -85,B 0,C 180,E1 -14616.427,E2 -14616.427} C_VEL
LIN {X 0,Y 338.489,Z 251.96,A -85,B 0,C 180,E1 -14617.526,E2 -14617.526} C_VEL
LIN {X 0,Y 335.497,Z 231.259,A -85,B 0,C 180,E1 -14618.278,E2 -14618.278} C_VEL
LIN {X 0,Y 336.147,Z 217.777,A -85,B 0,C 180,E1 -14621.509,E2 -14621.509} C_VEL
LIN {X 0,Y 335.904,Z 214.133,A -85,B 0,C 180,E1 -14622.436,E2 -14622.436} C_VEL
LIN {X 0,Y 333.684,Z 203.045,A -85,B 0,C 180,E1 -14625.456,E2 -14625.456} C_VEL
LIN {X 0,Y 333.646,Z 202.924,A -85,B 0,C 180,E1 -14629.315,E2 -14629.315} C_VEL
LIN {X 0,Y 333.664,Z 202.921,A -85,B 0,C 180,E1 -14633.167,E2 -14633.167} C_VEL
LIN {X 0,Y 333.638,Z 202.923,A -85,B 0,C 180,E1 -14636.791,E2 -14636.791} C_VEL
LIN {X 0,Y 333.701,Z 202.919,A -85,B 0,C 180,E1 -14639.709,E2 -14639.709} C_VEL
LIN {X 0,Y 333.742,Z 202.909,A -85,B 0,C 180,E1 -14642.4,E2 -14642.4} C_VEL
LIN {X 0,Y 333.725,Z 202.914,A -85,B 0,C 180,E1 -14645.09,E2 -14645.09} C_VEL
LIN {X 0,Y 333.681,Z 202.919,A -85,B 0,C 180,E1 -14649.019,E2 -14649.019} C_VEL
LIN {X 0,Y 333.793,Z 202.907,A -85,B 0,C 180,E1 -14651.589,E2 -14651.589} C_VEL
LIN {X 0,Y 333.806,Z 202.905,A -85,B 0,C 180,E1 -14655.576,E2 -14655.576} C_VEL
LIN {X 0,Y 333.832,Z 202.902,A -85,B 0,C 180,E1 -14659.077,E2 -14659.077} C_VEL
LIN {X 0,Y 334.023,Z 202.876,A -85,B 0,C 180,E1 -14662.747,E2 -14662.747} C_VEL
LIN {X 0,Y 333.809,Z 202.907,A -85,B 0,C 180,E1 -14665.168,E2 -14665.168} C_VEL
LIN {X 0,Y 334.104,Z 202.866,A -85,B 0,C 180,E1 -14667.588,E2 -14667.588} C_VEL
LIN {X 0,Y 334.245,Z 202.847,A -85,B 0,C 180,E1 -14669.999,E2 -14669.999} C_VEL
LIN {X 0,Y 334.104,Z 202.865,A -85,B 0,C 180,E1 -14672.41,E2 -14672.41} C_VEL
LIN {X 0,Y 334.011,Z 202.876,A -85,B 0,C 180,E1 -14676.038,E2 -14676.038} C_VEL
LIN {X 0,Y 333.981,Z 202.881,A -85,B 0,C 180,E1 -14678.5,E2 -14678.5} C_VEL
LIN {X 0,Y 333.787,Z 202.904,A -85,B 0,C 180,E1 -14682.154,E2 -14682.154} C_VEL
LIN {X 0,Y 333.773,Z 202.905,A -85,B 0,C 180,E1 -14685.885,E2 -14685.885} C_VEL
LIN {X 0,Y 333.792,Z 202.908,A -85,B 0,C 180,E1 -14688.655,E2 -14688.655} C_VEL
LIN {X 0,Y 333.687,Z 202.918,A -85,B 0,C 180,E1 -14692.277,E2 -14692.277} C_VEL
LIN {X 0,Y 333.73,Z 202.913,A -85,B 0,C 180,E1 -14696.245,E2 -14696.245} C_VEL
LIN {X 0,Y 333.705,Z 202.917,A -85,B 0,C 180,E1 -14698.971,E2 -14698.971} C_VEL
LIN {X 0,Y 333.639,Z 202.928,A -85,B 0,C 180,E1 -14702.587,E2 -14702.587} C_VEL
LIN {X 0,Y 333.671,Z 202.921,A -85,B 0,C 180,E1 -14706.138,E2 -14706.138} C_VEL
LIN {X 0,Y 333.677,Z 202.918,A -85,B 0,C 180,E1 -14709.186,E2 -14709.186} C_VEL
LIN {X 0,Y 333.687,Z 202.919,A -85,B 0,C 180,E1 -14710.6,E2 -14710.6} C_VEL
LIN {X 0,Y 333.068,Z 203.002,A -85,B 0,C 180,E1 -14711.607,E2 -14711.607} C_VEL
LIN {X 0,Y 330.183,Z 203.359,A -85,B 0,C 180,E1 -14713.243,E2 -14713.243} C_VEL
LIN {X 0,Y 327.71,Z 203.665,A -85,B 0,C 180,E1 -14714.57,E2 -14714.57} C_VEL
LIN {X 0,Y 326.657,Z 203.792,A -85,B 0,C 180,E1 -14715.597,E2 -14715.597} C_VEL
LIN {X 0,Y 326.579,Z 203.802,A -85,B 0,C 180,E1 -14715.946,E2 -14715.946} C_VEL
LIN {X 0,Y 326.596,Z 203.801,A -85,B 0,C 180,E1 -14719.793,E2 -14719.793} C_VEL
LIN {X 0,Y 326.625,Z 203.796,A -85,B 0,C 180,E1 -14722.953,E2 -14722.953} C_VEL
LIN {X 0,Y 326.615,Z 203.797,A -85,B 0,C 180,E1 -14727.052,E2 -14727.052} C_VEL
LIN {X 0,Y 326.654,Z 203.796,A -85,B 0,C 180,E1 -14730.341,E2 -14730.341} C_VEL
LIN {X 0,Y 326.682,Z 203.791,A -85,B 0,C 180,E1 -14734.516,E2 -14734.516} C_VEL
LIN {X 0,Y 326.638,Z 203.796,A -85,B 0,C 180,E1 -14738.545,E2 -14738.545} C_VEL
LIN {X 0,Y 326.736,Z 203.782,A -85,B 0,C 180,E1 -14741.178,E2 -14741.178} C_VEL
LIN {X 0,Y 326.755,Z 203.781,A -85,B 0,C 180,E1 -14745.433,E2 -14745.433} C_VEL
LIN {X 0,Y 326.762,Z 203.779,A -85,B 0,C 180,E1 -14748.839,E2 -14748.839} C_VEL
LIN {X 0,Y 326.95,Z 203.756,A -85,B 0,C 180,E1 -14752.59,E2 -14752.59} C_VEL
LIN {X 0,Y 326.768,Z 203.779,A -85,B 0,C 180,E1 -14755.065,E2 -14755.065} C_VEL
LIN {X 0,Y 327.038,Z 203.749,A -85,B 0,C 180,E1 -14757.537,E2 -14757.537} C_VEL
LIN {X 0,Y 327.191,Z 203.728,A -85,B 0,C 180,E1 -14760.001,E2 -14760.001} C_VEL
LIN {X 0,Y 327.038,Z 203.745,A -85,B 0,C 180,E1 -14762.464,E2 -14762.464} C_VEL
LIN {X 0,Y 326.988,Z 203.752,A -85,B 0,C 180,E1 -14766.17,E2 -14766.17} C_VEL
LIN {X 0,Y 326.908,Z 203.761,A -85,B 0,C 180,E1 -14768.656,E2 -14768.656} C_VEL
LIN {X 0,Y 326.727,Z 203.783,A -85,B 0,C 180,E1 -14772.422,E2 -14772.422} C_VEL
LIN {X 0,Y 326.748,Z 203.782,A -85,B 0,C 180,E1 -14774.958,E2 -14774.958} C_VEL
LIN {X 0,Y 326.726,Z 203.785,A -85,B 0,C 180,E1 -14778.839,E2 -14778.839} C_VEL
LIN {X 0,Y 326.615,Z 203.798,A -85,B 0,C 180,E1 -14782.788,E2 -14782.788} C_VEL
LIN {X 0,Y 326.685,Z 203.792,A -85,B 0,C 180,E1 -14785.485,E2 -14785.485} C_VEL
LIN {X 0,Y 326.643,Z 203.796,A -85,B 0,C 180,E1 -14789.661,E2 -14789.661} C_VEL
LIN {X 0,Y 326.602,Z 203.799,A -85,B 0,C 180,E1 -14794.021,E2 -14794.021} C_VEL
LIN {X 0,Y 326.623,Z 203.801,A -85,B 0,C 180,E1 -14797.24,E2 -14797.24} C_VEL
LIN {X 0,Y 326.574,Z 203.807,A -85,B 0,C 180,E1 -14801.133,E2 -14801.133} C_VEL
LIN {X 0,Y 326.524,Z 203.812,A -85,B 0,C 180,E1 -14804.744,E2 -14804.744} C_VEL
LIN {X 0,Y 326.573,Z 203.803,A -85,B 0,C 180,E1 -14808.155,E2 -14808.155} C_VEL
LIN {X 0,Y 326.595,Z 203.801,A -85,B 0,C 180,E1 -14811.389,E2 -14811.389} C_VEL
LIN {X 0,Y 326.618,Z 203.803,A -85,B 0,C 180,E1 -14814.853,E2 -14814.853} C_VEL
LIN {X 0,Y 326.674,Z 204.014,A -85,B 0,C 180,E1 -14816.757,E2 -14816.757} C_VEL
LIN {X 0,Y 330.3,Z 220.079,A -85,B 0,C 180,E1 -14820.352,E2 -14820.352} C_VEL
LIN {X 0,Y 332.277,Z 229.033,A -85,B 0,C 180,E1 -14822.27,E2 -14822.27} C_VEL
LIN {X 0,Y 332.254,Z 232.982,A -85,B 0,C 180,E1 -14823.056,E2 -14823.056} C_VEL
LIN {X 0,Y 329.495,Z 257.474,A -85,B 0,C 180,E1 -14827.754,E2 -14827.754} C_VEL
LIN {X 0,Y 329.303,Z 260.059,A -85,B 0,C 180,E1 -14828.194,E2 -14828.194} C_VEL
LIN {X 0,Y 332.263,Z 295.035,A -85,B 0,C 180,E1 -14829.257,E2 -14829.257} C_VEL
LIN {X 0,Y 330.86,Z 365.393,A -85,B 0,C 180,E1 -14831.06,E2 -14831.06} C_VEL
LIN {X 0,Y 330.178,Z 378.2,A -85,B 0,C 180,E1 -14831.623,E2 -14831.623} C_VEL
LIN {X 0,Y 329.488,Z 389.049,A -85,B 0,C 180,E1 -14832.306,E2 -14832.306} C_VEL
LIN {X 0,Y 328.726,Z 400.094,A -85,B 0,C 180,E1 -14833.226,E2 -14833.226} C_VEL
LIN {X 0,Y 327.783,Z 412.132,A -85,B 0,C 180,E1 -14834.519,E2 -14834.519} C_VEL
LIN {X 0,Y 326.969,Z 421.152,A -85,B 0,C 180,E1 -14835.731,E2 -14835.731} C_VEL
LIN {X 0,Y 326.283,Z 430.318,A -85,B 0,C 180,E1 -14837.246,E2 -14837.246} C_VEL
LIN {X 0,Y 325.696,Z 439.409,A -85,B 0,C 180,E1 -14839.118,E2 -14839.118} C_VEL
LIN {X 0,Y 325.414,Z 446.597,A -85,B 0,C 180,E1 -14840.993,E2 -14840.993} C_VEL
LIN {X 0,Y 325.396,Z 453.08,A -85,B 0,C 180,E1 -14843.179,E2 -14843.179} C_VEL
LIN {X 0,Y 325.361,Z 457.194,A -85,B 0,C 180,E1 -14845.044,E2 -14845.044} C_VEL
LIN {X 0,Y 325.513,Z 459.272,A -85,B 0,C 180,E1 -14846.287,E2 -14846.287} C_VEL
LIN {X 0,Y 325.64,Z 460.873,A -85,B 0,C 180,E1 -14847.527,E2 -14847.527} C_VEL
LIN {X 0,Y 325.631,Z 462.004,A -85,B 0,C 180,E1 -14848.764,E2 -14848.764} C_VEL
LIN {X 0,Y 325.595,Z 462.635,A -85,B 0,C 180,E1 -14850.001,E2 -14850.001} C_VEL
LIN {X 0,Y 325.607,Z 462.84,A -85,B 0,C 180,E1 -14851.238,E2 -14851.238} C_VEL
LIN {X 0,Y 325.454,Z 462.602,A -85,B 0,C 180,E1 -14852.476,E2 -14852.476} C_VEL
LIN {X 0,Y 325.263,Z 461.885,A -85,B 0,C 180,E1 -14853.717,E2 -14853.717} C_VEL
LIN {X 0,Y 325.214,Z 460.745,A -85,B 0,C 180,E1 -14854.96,E2 -14854.96} C_VEL
LIN {X 0,Y 325.204,Z 458.203,A -85,B 0,C 180,E1 -14856.827,E2 -14856.827} C_VEL
LIN {X 0,Y 325.281,Z 454.609,A -85,B 0,C 180,E1 -14858.7,E2 -14858.7} C_VEL
LIN {X 0,Y 325.594,Z 449.91,A -85,B 0,C 180,E1 -14860.573,E2 -14860.573} C_VEL
LIN {X 0,Y 326.351,Z 443.975,A -85,B 0,C 180,E1 -14862.437,E2 -14862.437} C_VEL
LIN {X 0,Y 327.38,Z 436.552,A -85,B 0,C 180,E1 -14864.293,E2 -14864.293} C_VEL
LIN {X 0,Y 328.756,Z 427.329,A -85,B 0,C 180,E1 -14866.136,E2 -14866.136} C_VEL
LIN {X 0,Y 330.244,Z 417.851,A -85,B 0,C 180,E1 -14867.654,E2 -14867.654} C_VEL
LIN {X 0,Y 331.946,Z 407.389,A -85,B 0,C 180,E1 -14868.998,E2 -14868.998} C_VEL
LIN {X 0,Y 333.583,Z 395.858,A -85,B 0,C 180,E1 -14870.182,E2 -14870.182} C_VEL
LIN {X 0,Y 335.111,Z 383.682,A -85,B 0,C 180,E1 -14871.129,E2 -14871.129} C_VEL
LIN {X 0,Y 336.526,Z 370.395,A -85,B 0,C 180,E1 -14871.88,E2 -14871.88} C_VEL
LIN {X 0,Y 337.412,Z 356.779,A -85,B 0,C 180,E1 -14872.383,E2 -14872.383} C_VEL
LIN {X 0,Y 339.686,Z 295.903,A -85,B 0,C 180,E1 -14874.038,E2 -14874.038} C_VEL
LIN {X 0,Y 337.997,Z 278.32,A -85,B 0,C 180,E1 -14874.796,E2 -14874.796} C_VEL
LIN {X 0,Y 335.296,Z 261.429,A -85,B 0,C 180,E1 -14875.669,E2 -14875.669} C_VEL
LIN {X 0,Y 334.461,Z 256.278,A -85,B 0,C 180,E1 -14875.989,E2 -14875.989} C_VEL
LIN {X 0,Y 336.862,Z 240.454,A -85,B 0,C 180,E1 -14879.017,E2 -14879.017} C_VEL
LIN {X 0,Y 335.945,Z 234.545,A -85,B 0,C 180,E1 -14880.418,E2 -14880.418} C_VEL
LIN {X 0,Y 333.66,Z 224.915,A -85,B 0,C 180,E1 -14882.947,E2 -14882.947} C_VEL
LIN {X 0,Y 330.802,Z 215.503,A -85,B 0,C 180,E1 -14885.749,E2 -14885.749} C_VEL
LIN {X 0,Y 327.987,Z 207.734,A -85,B 0,C 180,E1 -14888.419,E2 -14888.419} C_VEL
LIN {X 0,Y 326.579,Z 203.921,A -85,B 0,C 180,E1 -14889.936,E2 -14889.936} C_VEL
LIN {X 0,Y 326.564,Z 203.809,A -85,B 0,C 180,E1 -14893.526,E2 -14893.526} C_VEL
LIN {X 0,Y 326.579,Z 203.807,A -85,B 0,C 180,E1 -14897.028,E2 -14897.028} C_VEL
LIN {X 0,Y 326.615,Z 203.8,A -85,B 0,C 180,E1 -14900.773,E2 -14900.773} C_VEL
LIN {X 0,Y 326.615,Z 203.797,A -85,B 0,C 180,E1 -14904.48,E2 -14904.48} C_VEL
LIN {X 0,Y 326.611,Z 203.802,A -85,B 0,C 180,E1 -14907.455,E2 -14907.455} C_VEL
LIN {X 0,Y 326.651,Z 203.794,A -85,B 0,C 180,E1 -14910.339,E2 -14910.339} C_VEL
LIN {X 0,Y 326.693,Z 203.79,A -85,B 0,C 180,E1 -14914.516,E2 -14914.516} C_VEL
LIN {X 0,Y 326.649,Z 203.796,A -85,B 0,C 180,E1 -14918.545,E2 -14918.545} C_VEL
LIN {X 0,Y 326.748,Z 203.782,A -85,B 0,C 180,E1 -14921.177,E2 -14921.177} C_VEL
LIN {X 0,Y 326.766,Z 203.783,A -85,B 0,C 180,E1 -14925.433,E2 -14925.433} C_VEL
LIN {X 0,Y 326.787,Z 203.978,A -85,B 0,C 180,E1 -14926.869,E2 -14926.869} C_VEL
LIN {X 0,Y 329.772,Z 212.498,A -85,B 0,C 180,E1 -14930.183,E2 -14930.183} C_VEL
LIN {X 0,Y 331.56,Z 217.958,A -85,B 0,C 180,E1 -14932.08,E2 -14932.08} C_VEL
LIN {X 0,Y 333.698,Z 226.643,A -85,B 0,C 180,E1 -14934.779,E2 -14934.779} C_VEL
LIN {X 0,Y 334.872,Z 232.214,A -85,B 0,C 180,E1 -14936.39,E2 -14936.39} C_VEL
LIN {X 0,Y 334.702,Z 235.081,A -85,B 0,C 180,E1 -14937.028,E2 -14937.028} C_VEL
LIN {X 0,Y 338.401,Z 249.798,A -85,B 0,C 180,E1 -14938.063,E2 -14938.063} C_VEL
LIN {X 0,Y 340.547,Z 260.483,A -85,B 0,C 180,E1 -14938.706,E2 -14938.706} C_VEL
LIN {X 0,Y 337.424,Z 321.891,A -85,B 0,C 180,E1 -14940.697,E2 -14940.697} C_VEL
LIN {X 0,Y 336.721,Z 334.388,A -85,B 0,C 180,E1 -14941.345,E2 -14941.345} C_VEL
LIN {X 0,Y 335.691,Z 346.608,A -85,B 0,C 180,E1 -14942.249,E2 -14942.249} C_VEL
LIN {X 0,Y 334.52,Z 357.335,A -85,B 0,C 180,E1 -14943.312,E2 -14943.312} C_VEL
LIN {X 0,Y 333.189,Z 367.467,A -85,B 0,C 180,E1 -14944.599,E2 -14944.599} C_VEL
LIN {X 0,Y 331.814,Z 376.607,A -85,B 0,C 180,E1 -14946.079,E2 -14946.079} C_VEL
LIN {X 0,Y 330.534,Z 384.152,A -85,B 0,C 180,E1 -14947.636,E2 -14947.636} C_VEL
LIN {X 0,Y 329.387,Z 390.256,A -85,B 0,C 180,E1 -14949.208,E2 -14949.208} C_VEL
LIN {X 0,Y 328.262,Z 395.87,A -85,B 0,C 180,E1 -14951.109,E2 -14951.109} C_VEL
LIN {X 0,Y 327.325,Z 399.974,A -85,B 0,C 180,E1 -14953.028,E2 -14953.028} C_VEL
LIN {X 0,Y 326.624,Z 402.644,A -85,B 0,C 180,E1 -14954.963,E2 -14954.963} C_VEL
LIN {X 0,Y 326.256,Z 403.71,A -85,B 0,C 180,E1 -14956.262,E2 -14956.262} C_VEL
LIN {X 0,Y 325.833,Z 404.213,A -85,B 0,C 180,E1 -14958.367,E2 -14958.367} C_VEL
LIN {X 0,Y 325.608,Z 403.444,A -85,B 0,C 180,E1 -14960.202,E2 -14960.202} C_VEL
LIN {X 0,Y 325.573,Z 401.778,A -85,B 0,C 180,E1 -14961.84,E2 -14961.84} C_VEL
LIN {X 0,Y 325.712,Z 399.065,A -85,B 0,C 180,E1 -14963.526,E2 -14963.526} C_VEL
LIN {X 0,Y 326.012,Z 394.423,A -85,B 0,C 180,E1 -14965.54,E2 -14965.54} C_VEL
LIN {X 0,Y 326.391,Z 388.3,A -85,B 0,C 180,E1 -14967.468,E2 -14967.468} C_VEL
LIN {X 0,Y 326.744,Z 382.349,A -85,B 0,C 180,E1 -14968.943,E2 -14968.943} C_VEL
LIN {X 0,Y 327.367,Z 374.031,A -85,B 0,C 180,E1 -14970.583,E2 -14970.583} C_VEL
LIN {X 0,Y 328.027,Z 364.846,A -85,B 0,C 180,E1 -14972.023,E2 -14972.023} C_VEL
LIN {X 0,Y 328.61,Z 355.195,A -85,B 0,C 180,E1 -14973.232,E2 -14973.232} C_VEL
LIN {X 0,Y 329.2,Z 344.672,A -85,B 0,C 180,E1 -14974.268,E2 -14974.268} C_VEL
LIN {X 0,Y 329.719,Z 333.163,A -85,B 0,C 180,E1 -14975.134,E2 -14975.134} C_VEL
LIN {X 0,Y 330.113,Z 320.252,A -85,B 0,C 180,E1 -14975.819,E2 -14975.819} C_VEL
LIN {X 0,Y 330.513,Z 301.201,A -85,B 0,C 180,E1 -14976.414,E2 -14976.414} C_VEL
LIN {X 0,Y 331.668,Z 253.367,A -85,B 0,C 180,E1 -14977.761,E2 -14977.761} C_VEL
LIN {X 0,Y 328.517,Z 231.649,A -85,B 0,C 180,E1 -14978.552,E2 -14978.552} C_VEL
LIN {X 0,Y 329.181,Z 218.861,A -85,B 0,C 180,E1 -14981.647,E2 -14981.647} C_VEL
LIN {X 0,Y 328.666,Z 214.008,A -85,B 0,C 180,E1 -14982.914,E2 -14982.914} C_VEL
LIN {X 0,Y 326.63,Z 203.984,A -85,B 0,C 180,E1 -14985.679,E2 -14985.679} C_VEL
LIN {X 0,Y 326.591,Z 203.805,A -85,B 0,C 180,E1 -14989.79,E2 -14989.79} C_VEL
LIN {X 0,Y 326.629,Z 203.796,A -85,B 0,C 180,E1 -14992.952,E2 -14992.952} C_VEL
LIN {X 0,Y 326.607,Z 203.801,A -85,B 0,C 180,E1 -14995.98,E2 -14995.98} C_VEL
LIN {X 0,Y 326.659,Z 203.792,A -85,B 0,C 180,E1 -15000.34,E2 -15000.34} C_VEL
LIN {X 0,Y 326.689,Z 203.788,A -85,B 0,C 180,E1 -15004.515,E2 -15004.515} C_VEL
LIN {X 0,Y 326.645,Z 203.794,A -85,B 0,C 180,E1 -15008.545,E2 -15008.545} C_VEL
LIN {X 0,Y 326.743,Z 203.785,A -85,B 0,C 180,E1 -15011.177,E2 -15011.177} C_VEL
LIN {X 0,Y 326.761,Z 203.784,A -85,B 0,C 180,E1 -15015.432,E2 -15015.432} C_VEL
LIN {X 0,Y 326.768,Z 203.78,A -85,B 0,C 180,E1 -15018.838,E2 -15018.838} C_VEL
LIN {X 0,Y 326.977,Z 203.753,A -85,B 0,C 180,E1 -15022.59,E2 -15022.59} C_VEL
LIN {X 0,Y 326.776,Z 203.782,A -85,B 0,C 180,E1 -15025.064,E2 -15025.064} C_VEL
LIN {X 0,Y 327.045,Z 203.746,A -85,B 0,C 180,E1 -15027.536,E2 -15027.536} C_VEL
LIN {X 0,Y 327.196,Z 203.725,A -85,B 0,C 180,E1 -15029.999,E2 -15029.999} C_VEL
LIN {X 0,Y 327.045,Z 203.745,A -85,B 0,C 180,E1 -15032.462,E2 -15032.462} C_VEL
LIN {X 0,Y 326.986,Z 203.751,A -85,B 0,C 180,E1 -15036.168,E2 -15036.168} C_VEL
LIN {X 0,Y 326.911,Z 203.763,A -85,B 0,C 180,E1 -15038.654,E2 -15038.654} C_VEL
LIN {X 0,Y 326.731,Z 203.784,A -85,B 0,C 180,E1 -15042.42,E2 -15042.42} C_VEL
LIN {X 0,Y 326.75,Z 203.785,A -85,B 0,C 180,E1 -15044.957,E2 -15044.957} C_VEL
LIN {X 0,Y 326.729,Z 203.788,A -85,B 0,C 180,E1 -15048.838,E2 -15048.838} C_VEL
LIN {X 0,Y 326.615,Z 203.802,A -85,B 0,C 180,E1 -15052.787,E2 -15052.787} C_VEL
LIN {X 0,Y 326.684,Z 203.789,A -85,B 0,C 180,E1 -15055.483,E2 -15055.483} C_VEL
LIN {X 0,Y 326.654,Z 203.792,A -85,B 0,C 180,E1 -15059.658,E2 -15059.658} C_VEL
LIN {X 0,Y 326.602,Z 203.8,A -85,B 0,C 180,E1 -15064.019,E2 -15064.019} C_VEL
LIN {X 0,Y 326.623,Z 203.797,A -85,B 0,C 180,E1 -15067.239,E2 -15067.239} C_VEL
LIN {X 0,Y 326.615,Z 203.798,A -85,B 0,C 180,E1 -15070.597,E2 -15070.597} C_VEL
LIN {X 0,Y 326.615,Z 203.797,A -85,B 0,C 180,E1 -15073.515,E2 -15073.515} C_VEL
LIN {X 0,Y 326.579,Z 203.802,A -85,B 0,C 180,E1 -15075.946,E2 -15075.946} C_VEL
LIN {X 0,Y 325.926,Z 203.887,A -85,B 0,C 180,E1 -15076.974,E2 -15076.974} C_VEL
LIN {X 0,Y 323.066,Z 204.243,A -85,B 0,C 180,E1 -15078.647,E2 -15078.647} C_VEL
LIN {X 0,Y 320.645,Z 204.544,A -85,B 0,C 180,E1 -15080.002,E2 -15080.002} C_VEL
LIN {X 0,Y 319.627,Z 204.668,A -85,B 0,C 180,E1 -15081.052,E2 -15081.052} C_VEL
LIN {X 0,Y 319.555,Z 204.677,A -85,B 0,C 180,E1 -15081.408,E2 -15081.408} C_VEL
LIN {X 0,Y 319.553,Z 204.677,A -85,B 0,C 180,E1 -15085.123,E2 -15085.123} C_VEL
LIN {X 0,Y 319.567,Z 204.675,A -85,B 0,C 180,E1 -15089.056,E2 -15089.056} C_VEL
LIN {X 0,Y 319.601,Z 204.673,A -85,B 0,C 180,E1 -15092.498,E2 -15092.498} C_VEL
LIN {X 0,Y 319.596,Z 204.672,A -85,B 0,C 180,E1 -15095.304,E2 -15095.304} C_VEL
LIN {X 0,Y 319.589,Z 204.678,A -85,B 0,C 180,E1 -15098.048,E2 -15098.048} C_VEL
LIN {X 0,Y 319.681,Z 204.661,A -85,B 0,C 180,E1 -15100.962,E2 -15100.962} C_VEL
LIN {X 0,Y 319.723,Z 204.656,A -85,B 0,C 180,E1 -15105.276,E2 -15105.276} C_VEL
LIN {X 0,Y 319.745,Z 204.658,A -85,B 0,C 180,E1 -15109.873,E2 -15109.873} C_VEL
LIN {X 0,Y 319.905,Z 204.634,A -85,B 0,C 180,E1 -15112.426,E2 -15112.426} C_VEL
LIN {X 0,Y 319.738,Z 204.654,A -85,B 0,C 180,E1 -15114.957,E2 -15114.957} C_VEL
LIN {X 0,Y 319.982,Z 204.627,A -85,B 0,C 180,E1 -15117.483,E2 -15117.483} C_VEL
LIN {X 0,Y 320.143,Z 204.606,A -85,B 0,C 180,E1 -15120.001,E2 -15120.001} C_VEL
LIN {X 0,Y 319.982,Z 204.623,A -85,B 0,C 180,E1 -15122.518,E2 -15122.518} C_VEL
LIN {X 0,Y 319.943,Z 204.629,A -85,B 0,C 180,E1 -15126.306,E2 -15126.306} C_VEL
LIN {X 0,Y 319.836,Z 204.642,A -85,B 0,C 180,E1 -15128.849,E2 -15128.849} C_VEL
LIN {X 0,Y 319.675,Z 204.662,A -85,B 0,C 180,E1 -15132.701,E2 -15132.701} C_VEL
LIN {X 0,Y 319.693,Z 204.664,A -85,B 0,C 180,E1 -15135.296,E2 -15135.296} C_VEL
LIN {X 0,Y 319.669,Z 204.667,A -85,B 0,C 180,E1 -15139.256,E2 -15139.256} C_VEL
LIN {X 0,Y 319.565,Z 204.681,A -85,B 0,C 180,E1 -15143.32,E2 -15143.32} C_VEL
LIN {X 0,Y 319.613,Z 204.67,A -85,B 0,C 180,E1 -15146.091,E2 -15146.091} C_VEL
LIN {X 0,Y 319.575,Z 204.677,A -85,B 0,C 180,E1 -15148.936,E2 -15148.936} C_VEL
LIN {X 0,Y 319.526,Z 204.681,A -85,B 0,C 180,E1 -15151.863,E2 -15151.863} C_VEL
LIN {X 0,Y 319.575,Z 204.676,A -85,B 0,C 180,E1 -15155.544,E2 -15155.544} C_VEL
LIN {X 0,Y 319.555,Z 204.678,A -85,B 0,C 180,E1 -15159.67,E2 -15159.67} C_VEL
LIN {X 0,Y 319.518,Z 204.683,A -85,B 0,C 180,E1 -15163.462,E2 -15163.462} C_VEL
LIN {X 0,Y 319.551,Z 204.682,A -85,B 0,C 180,E1 -15167.018,E2 -15167.018} C_VEL
LIN {X 0,Y 319.544,Z 204.68,A -85,B 0,C 180,E1 -15170.372,E2 -15170.372} C_VEL
LIN {X 0,Y 319.578,Z 204.677,A -85,B 0,C 180,E1 -15174.458,E2 -15174.458} C_VEL
LIN {X 0,Y 319.609,Z 204.855,A -85,B 0,C 180,E1 -15176.405,E2 -15176.405} C_VEL
LIN {X 0,Y 322.736,Z 218.661,A -85,B 0,C 180,E1 -15179.584,E2 -15179.584} C_VEL
LIN {X 0,Y 325.396,Z 231.144,A -85,B 0,C 180,E1 -15182.318,E2 -15182.318} C_VEL
LIN {X 0,Y 324.529,Z 239.596,A -85,B 0,C 180,E1 -15183.991,E2 -15183.991} C_VEL
LIN {X 0,Y 322.347,Z 259.451,A -85,B 0,C 180,E1 -15187.867,E2 -15187.867} C_VEL
LIN {X 0,Y 324.75,Z 288.375,A -85,B 0,C 180,E1 -15188.792,E2 -15188.792} C_VEL
LIN {X 0,Y 325.293,Z 296.104,A -85,B 0,C 180,E1 -15189.025,E2 -15189.025} C_VEL
LIN {X 0,Y 323.877,Z 364.979,A -85,B 0,C 180,E1 -15190.841,E2 -15190.841} C_VEL
LIN {X 0,Y 323.251,Z 377.012,A -85,B 0,C 180,E1 -15191.379,E2 -15191.379} C_VEL
LIN {X 0,Y 322.44,Z 389.067,A -85,B 0,C 180,E1 -15192.152,E2 -15192.152} C_VEL
LIN {X 0,Y 321.628,Z 400.772,A -85,B 0,C 180,E1 -15193.171,E2 -15193.171} C_VEL
LIN {X 0,Y 320.7,Z 412.056,A -85,B 0,C 180,E1 -15194.429,E2 -15194.429} C_VEL
LIN {X 0,Y 319.867,Z 421.527,A -85,B 0,C 180,E1 -15195.755,E2 -15195.755} C_VEL
LIN {X 0,Y 319.182,Z 430.393,A -85,B 0,C 180,E1 -15197.281,E2 -15197.281} C_VEL
LIN {X 0,Y 318.694,Z 437.985,A -85,B 0,C 180,E1 -15198.875,E2 -15198.875} C_VEL
LIN {X 0,Y 318.35,Z 445.365,A -85,B 0,C 180,E1 -15200.791,E2 -15200.791} C_VEL
LIN {X 0,Y 318.299,Z 450.29,A -85,B 0,C 180,E1 -15202.388,E2 -15202.388} C_VEL
LIN {X 0,Y 318.369,Z 454.952,A -85,B 0,C 180,E1 -15204.3,E2 -15204.3} C_VEL
LIN {X 0,Y 318.433,Z 458.363,A -85,B 0,C 180,E1 -15206.205,E2 -15206.205} C_VEL
LIN {X 0,Y 318.566,Z 460.009,A -85,B 0,C 180,E1 -15207.472,E2 -15207.472} C_VEL
LIN {X 0,Y 318.588,Z 461.194,A -85,B 0,C 180,E1 -15208.737,E2 -15208.737} C_VEL
LIN {X 0,Y 318.551,Z 461.896,A -85,B 0,C 180,E1 -15210.001,E2 -15210.001} C_VEL
LIN {X 0,Y 318.558,Z 462.137,A -85,B 0,C 180,E1 -15211.265,E2 -15211.265} C_VEL
LIN {X 0,Y 318.385,Z 461.934,A -85,B 0,C 180,E1 -15212.531,E2 -15212.531} C_VEL
LIN {X 0,Y 318.175,Z 461.284,A -85,B 0,C 180,E1 -15213.8,E2 -15213.8} C_VEL
LIN {X 0,Y 318.128,Z 458.839,A -85,B 0,C 180,E1 -15216.207,E2 -15216.207} C_VEL
LIN {X 0,Y 318.164,Z 455.511,A -85,B 0,C 180,E1 -15218.256,E2 -15218.256} C_VEL
LIN {X 0,Y 318.42,Z 451.278,A -85,B 0,C 180,E1 -15220.171,E2 -15220.171} C_VEL
LIN {X 0,Y 319.078,Z 445.868,A -85,B 0,C 180,E1 -15222.079,E2 -15222.079} C_VEL
LIN {X 0,Y 320.018,Z 439.059,A -85,B 0,C 180,E1 -15223.98,E2 -15223.98} C_VEL
LIN {X 0,Y 321.522,Z 430.098,A -85,B 0,C 180,E1 -15225.976,E2 -15225.976} C_VEL
LIN {X 0,Y 322.808,Z 422.122,A -85,B 0,C 180,E1 -15227.42,E2 -15227.42} C_VEL
LIN {X 0,Y 324.628,Z 411.615,A -85,B 0,C 180,E1 -15228.951,E2 -15228.951} C_VEL
LIN {X 0,Y 326.512,Z 399.828,A -85,B 0,C 180,E1 -15230.31,E2 -15230.31} C_VEL
LIN {X 0,Y 328.192,Z 388.029,A -85,B 0,C 180,E1 -15231.349,E2 -15231.349} C_VEL
LIN {X 0,Y 329.697,Z 375.934,A -85,B 0,C 180,E1 -15232.151,E2 -15232.151} C_VEL
LIN {X 0,Y 330.823,Z 362.769,A -85,B 0,C 180,E1 -15232.771,E2 -15232.771} C_VEL
LIN {X 0,Y 331.952,Z 337.462,A -85,B 0,C 180,E1 -15233.514,E2 -15233.514} C_VEL
LIN {X 0,Y 333.63,Z 296.114,A -85,B 0,C 180,E1 -15234.683,E2 -15234.683} C_VEL
LIN {X 0,Y 331.882,Z 278.361,A -85,B 0,C 180,E1 -15235.482,E2 -15235.482} C_VEL
LIN {X 0,Y 329.2,Z 261.475,A -85,B 0,C 180,E1 -15236.409,E2 -15236.409} C_VEL
LIN {X 0,Y 328.245,Z 255.911,A -85,B 0,C 180,E1 -15236.763,E2 -15236.763} C_VEL
LIN {X 0,Y 330.337,Z 242.953,A -85,B 0,C 180,E1 -15239.297,E2 -15239.297} C_VEL
LIN {X 0,Y 330.094,Z 239.88,A -85,B 0,C 180,E1 -15240.023,E2 -15240.023} C_VEL
LIN {X 0,Y 328.13,Z 230.928,A -85,B 0,C 180,E1 -15242.376,E2 -15242.376} C_VEL
LIN {X 0,Y 325.779,Z 222.186,A -85,B 0,C 180,E1 -15244.937,E2 -15244.937} C_VEL
LIN {X 0,Y 322.99,Z 213.868,A -85,B 0,C 180,E1 -15247.738,E2 -15247.738} C_VEL
LIN {X 0,Y 320.826,Z 208.183,A -85,B 0,C 180,E1 -15249.94,E2 -15249.94} C_VEL
LIN {X 0,Y 319.518,Z 204.782,A -85,B 0,C 180,E1 -15251.489,E2 -15251.489} C_VEL
LIN {X 0,Y 319.491,Z 204.687,A -85,B 0,C 180,E1 -15254.743,E2 -15254.743} C_VEL
LIN {X 0,Y 319.529,Z 204.68,A -85,B 0,C 180,E1 -15258.403,E2 -15258.403} C_VEL
LIN {X 0,Y 319.546,Z 204.677,A -85,B 0,C 180,E1 -15261.988,E2 -15261.988} C_VEL
LIN {X 0,Y 319.564,Z 204.68,A -85,B 0,C 180,E1 -15265.123,E2 -15265.123} C_VEL
LIN {X 0,Y 319.569,Z 204.675,A -85,B 0,C 180,E1 -15269.059,E2 -15269.059} C_VEL
LIN {X 0,Y 319.609,Z 204.671,A -85,B 0,C 180,E1 -15272.498,E2 -15272.498} C_VEL
LIN {X 0,Y 319.608,Z 204.67,A -85,B 0,C 180,E1 -15275.304,E2 -15275.304} C_VEL
LIN {X 0,Y 319.6,Z 204.675,A -85,B 0,C 180,E1 -15278.047,E2 -15278.047} C_VEL
LIN {X 0,Y 319.692,Z 204.661,A -85,B 0,C 180,E1 -15280.962,E2 -15280.962} C_VEL
LIN {X 0,Y 319.753,Z 204.783,A -85,B 0,C 180,E1 -15285.316,E2 -15285.316} C_VEL
LIN {X 0,Y 321.931,Z 210.945,A -85,B 0,C 180,E1 -15288.03,E2 -15288.03} C_VEL
LIN {X 0,Y 324.935,Z 219.529,A -85,B 0,C 180,E1 -15291.291,E2 -15291.291} C_VEL
LIN {X 0,Y 327.069,Z 228.173,A -85,B 0,C 180,E1 -15294.116,E2 -15294.116} C_VEL
LIN {X 0,Y 328.424,Z 234.431,A -85,B 0,C 180,E1 -15296.011,E2 -15296.011} C_VEL
LIN {X 0,Y 328.586,Z 235.804,A -85,B 0,C 180,E1 -15296.263,E2 -15296.263} C_VEL
LIN {X 0,Y 332.468,Z 251.15,A -85,B 0,C 180,E1 -15297.406,E2 -15297.406} C_VEL
LIN {X 0,Y 334.549,Z 261.79,A -85,B 0,C 180,E1 -15298.078,E2 -15298.078} C_VEL
LIN {X 0,Y 331.36,Z 321.183,A -85,B 0,C 180,E1 -15300.037,E2 -15300.037} C_VEL
LIN {X 0,Y 330.605,Z 334.052,A -85,B 0,C 180,E1 -15300.701,E2 -15300.701} C_VEL
LIN {X 0,Y 329.597,Z 345.35,A -85,B 0,C 180,E1 -15301.527,E2 -15301.527} C_VEL
LIN {X 0,Y 328.331,Z 356.497,A -85,B 0,C 180,E1 -15302.606,E2 -15302.606} C_VEL
LIN {X 0,Y 327.045,Z 366.459,A -85,B 0,C 180,E1 -15303.85,E2 -15303.85} C_VEL
LIN {X 0,Y 325.866,Z 373.662,A -85,B 0,C 180,E1 -15304.948,E2 -15304.948} C_VEL
LIN {X 0,Y 324.439,Z 381.964,A -85,B 0,C 180,E1 -15306.53,E2 -15306.53} C_VEL
LIN {X 0,Y 323.168,Z 388.632,A -85,B 0,C 180,E1 -15308.126,E2 -15308.126} C_VEL
LIN {X 0,Y 321.851,Z 394.814,A -85,B 0,C 180,E1 -15310.06,E2 -15310.06} C_VEL
LIN {X 0,Y 320.8,Z 399.395,A -85,B 0,C 180,E1 -15312.012,E2 -15312.012} C_VEL
LIN {X 0,Y 319.926,Z 402.57,A -85,B 0,C 180,E1 -15313.983,E2 -15313.983} C_VEL
LIN {X 0,Y 319.47,Z 403.934,A -85,B 0,C 180,E1 -15315.306,E2 -15315.306} C_VEL
LIN {X 0,Y 319.107,Z 404.737,A -85,B 0,C 180,E1 -15316.637,E2 -15316.637} C_VEL
LIN {X 0,Y 318.747,Z 404.852,A -85,B 0,C 180,E1 -15318.539,E2 -15318.539} C_VEL
LIN {X 0,Y 318.504,Z 403.617,A -85,B 0,C 180,E1 -15320.673,E2 -15320.673} C_VEL
LIN {X 0,Y 318.552,Z 401.025,A -85,B 0,C 180,E1 -15322.71,E2 -15322.71} C_VEL
LIN {X 0,Y 318.795,Z 396.976,A -85,B 0,C 180,E1 -15324.762,E2 -15324.762} C_VEL
LIN {X 0,Y 319.182,Z 391.175,A -85,B 0,C 180,E1 -15326.832,E2 -15326.832} C_VEL
LIN {X 0,Y 319.557,Z 384.676,A -85,B 0,C 180,E1 -15328.593,E2 -15328.593} C_VEL
LIN {X 0,Y 320.174,Z 376.558,A -85,B 0,C 180,E1 -15330.322,E2 -15330.322} C_VEL
LIN {X 0,Y 320.827,Z 367.109,A -85,B 0,C 180,E1 -15331.902,E2 -15331.902} C_VEL
LIN {X 0,Y 321.507,Z 356.712,A -85,B 0,C 180,E1 -15333.268,E2 -15333.268} C_VEL
LIN {X 0,Y 322.149,Z 346.235,A -85,B 0,C 180,E1 -15334.348,E2 -15334.348} C_VEL
LIN {X 0,Y 322.681,Z 334.811,A -85,B 0,C 180,E1 -15335.251,E2 -15335.251} C_VEL
LIN {X 0,Y 323.118,Z 322.635,A -85,B 0,C 180,E1 -15335.938,E2 -15335.938} C_VEL
LIN {X 0,Y 323.335,Z 309.294,A -85,B 0,C 180,E1 -15336.421,E2 -15336.421} C_VEL
LIN {X 0,Y 324.668,Z 253.559,A -85,B 0,C 180,E1 -15338.035,E2 -15338.035} C_VEL
LIN {X 0,Y 321.596,Z 232.073,A -85,B 0,C 180,E1 -15338.838,E2 -15338.838} C_VEL
LIN {X 0,Y 321.624,Z 229.767,A -85,B 0,C 180,E1 -15339.323,E2 -15339.323} C_VEL
LIN {X 0,Y 322.199,Z 218.621,A -85,B 0,C 180,E1 -15342.129,E2 -15342.129} C_VEL
LIN {X 0,Y 320.408,Z 208.767,A -85,B 0,C 180,E1 -15344.812,E2 -15344.812} C_VEL
LIN {X 0,Y 319.577,Z 204.843,A -85,B 0,C 180,E1 -15345.963,E2 -15345.963} C_VEL
LIN {X 0,Y 319.527,Z 204.683,A -85,B 0,C 180,E1 -15348.711,E2 -15348.711} C_VEL
LIN {X 0,Y 319.56,Z 204.677,A -85,B 0,C 180,E1 -15352.347,E2 -15352.347} C_VEL
LIN {X 0,Y 319.559,Z 204.678,A -85,B 0,C 180,E1 -15355.123,E2 -15355.123} C_VEL
LIN {X 0,Y 319.569,Z 204.676,A -85,B 0,C 180,E1 -15359.057,E2 -15359.057} C_VEL
LIN {X 0,Y 319.607,Z 204.67,A -85,B 0,C 180,E1 -15362.497,E2 -15362.497} C_VEL
LIN {X 0,Y 319.604,Z 204.675,A -85,B 0,C 180,E1 -15365.303,E2 -15365.303} C_VEL
LIN {X 0,Y 319.596,Z 204.672,A -85,B 0,C 180,E1 -15368.047,E2 -15368.047} C_VEL
LIN {X 0,Y 319.688,Z 204.662,A -85,B 0,C 180,E1 -15370.961,E2 -15370.961} C_VEL
LIN {X 0,Y 319.729,Z 204.66,A -85,B 0,C 180,E1 -15375.275,E2 -15375.275} C_VEL
LIN {X 0,Y 319.756,Z 204.652,A -85,B 0,C 180,E1 -15379.872,E2 -15379.872} C_VEL
LIN {X 0,Y 319.931,Z 204.63,A -85,B 0,C 180,E1 -15382.425,E2 -15382.425} C_VEL
LIN {X 0,Y 319.746,Z 204.657,A -85,B 0,C 180,E1 -15384.955,E2 -15384.955} C_VEL
LIN {X 0,Y 319.989,Z 204.625,A -85,B 0,C 180,E1 -15387.482,E2 -15387.482} C_VEL
LIN {X 0,Y 320.148,Z 204.603,A -85,B 0,C 180,E1 -15389.999,E2 -15389.999} C_VEL
LIN {X 0,Y 319.988,Z 204.624,A -85,B 0,C 180,E1 -15392.517,E2 -15392.517} C_VEL
LIN {X 0,Y 319.941,Z 204.629,A -85,B 0,C 180,E1 -15396.305,E2 -15396.305} C_VEL
LIN {X 0,Y 319.839,Z 204.646,A -85,B 0,C 180,E1 -15398.847,E2 -15398.847} C_VEL
LIN {X 0,Y 319.678,Z 204.665,A -85,B 0,C 180,E1 -15402.699,E2 -15402.699} C_VEL
LIN {X 0,Y 319.695,Z 204.661,A -85,B 0,C 180,E1 -15405.295,E2 -15405.295} C_VEL
LIN {X 0,Y 319.67,Z 204.664,A -85,B 0,C 180,E1 -15409.254,E2 -15409.254} C_VEL
LIN {X 0,Y 319.565,Z 204.676,A -85,B 0,C 180,E1 -15413.319,E2 -15413.319} C_VEL
LIN {X 0,Y 319.629,Z 204.668,A -85,B 0,C 180,E1 -15416.087,E2 -15416.087} C_VEL
LIN {X 0,Y 319.583,Z 204.676,A -85,B 0,C 180,E1 -15418.933,E2 -15418.933} C_VEL
LIN {X 0,Y 319.527,Z 204.681,A -85,B 0,C 180,E1 -15421.861,E2 -15421.861} C_VEL
LIN {X 0,Y 319.574,Z 204.674,A -85,B 0,C 180,E1 -15425.543,E2 -15425.543} C_VEL
LIN {X 0,Y 319.593,Z 204.674,A -85,B 0,C 180,E1 -15428.004,E2 -15428.004} C_VEL
LIN {X 0,Y 319.59,Z 204.672,A -85,B 0,C 180,E1 -15431.611,E2 -15431.611} C_VEL
LIN {X 0,Y 319.571,Z 204.675,A -85,B 0,C 180,E1 -15435.273,E2 -15435.273} C_VEL
LIN {X 0,Y 319.539,Z 204.681,A -85,B 0,C 180,E1 -15438.714,E2 -15438.714} C_VEL
LIN {X 0,Y 319.555,Z 204.677,A -85,B 0,C 180,E1 -15441.408,E2 -15441.408} C_VEL
LIN {X 0,Y 318.913,Z 204.76,A -85,B 0,C 180,E1 -15442.459,E2 -15442.459} C_VEL
LIN {X 0,Y 316.053,Z 205.118,A -85,B 0,C 180,E1 -15444.169,E2 -15444.169} C_VEL
LIN {X 0,Y 313.615,Z 205.42,A -85,B 0,C 180,E1 -15445.555,E2 -15445.555} C_VEL
LIN {X 0,Y 312.574,Z 205.549,A -85,B 0,C 180,E1 -15446.629,E2 -15446.629} C_VEL
LIN {X 0,Y 312.493,Z 205.557,A -85,B 0,C 180,E1 -15446.992,E2 -15446.992} C_VEL
LIN {X 0,Y 312.539,Z 205.554,A -85,B 0,C 180,E1 -15450.35,E2 -15450.35} C_VEL
LIN {X 0,Y 312.595,Z 205.549,A -85,B 0,C 180,E1 -15454.064,E2 -15454.064} C_VEL
LIN {X 0,Y 312.579,Z 205.547,A -85,B 0,C 180,E1 -15457.529,E2 -15457.529} C_VEL
LIN {X 0,Y 312.631,Z 205.542,A -85,B 0,C 180,E1 -15461.657,E2 -15461.657} C_VEL
LIN {X 0,Y 312.686,Z 205.536,A -85,B 0,C 180,E1 -15465.686,E2 -15465.686} C_VEL
LIN {X 0,Y 312.691,Z 205.536,A -85,B 0,C 180,E1 -15469.642,E2 -15469.642} C_VEL
LIN {X 0,Y 312.846,Z 205.514,A -85,B 0,C 180,E1 -15472.254,E2 -15472.254} C_VEL
LIN {X 0,Y 312.708,Z 205.53,A -85,B 0,C 180,E1 -15474.843,E2 -15474.843} C_VEL
LIN {X 0,Y 312.983,Z 205.495,A -85,B 0,C 180,E1 -15478.714,E2 -15478.714} C_VEL
LIN {X 0,Y 312.983,Z 205.498,A -85,B 0,C 180,E1 -15481.287,E2 -15481.287} C_VEL
LIN {X 0,Y 312.709,Z 205.531,A -85,B 0,C 180,E1 -15485.158,E2 -15485.158} C_VEL
LIN {X 0,Y 312.864,Z 205.514,A -85,B 0,C 180,E1 -15487.747,E2 -15487.747} C_VEL
LIN {X 0,Y 312.662,Z 205.539,A -85,B 0,C 180,E1 -15491.672,E2 -15491.672} C_VEL
LIN {X 0,Y 312.694,Z 205.533,A -85,B 0,C 180,E1 -15494.888,E2 -15494.888} C_VEL
LIN {X 0,Y 312.624,Z 205.544,A -85,B 0,C 180,E1 -15499.237,E2 -15499.237} C_VEL
LIN {X 0,Y 312.54,Z 205.552,A -85,B 0,C 180,E1 -15502.79,E2 -15502.79} C_VEL
LIN {X 0,Y 312.591,Z 205.545,A -85,B 0,C 180,E1 -15505.934,E2 -15505.934} C_VEL
LIN {X 0,Y 312.533,Z 205.553,A -85,B 0,C 180,E1 -15509.652,E2 -15509.652} C_VEL
LIN {X 0,Y 312.515,Z 205.555,A -85,B 0,C 180,E1 -15513.69,E2 -15513.69} C_VEL
LIN {X 0,Y 312.516,Z 205.557,A -85,B 0,C 180,E1 -15517.387,E2 -15517.387} C_VEL
LIN {X 0,Y 312.486,Z 205.56,A -85,B 0,C 180,E1 -15520.71,E2 -15520.71} C_VEL
LIN {X 0,Y 312.448,Z 205.562,A -85,B 0,C 180,E1 -15524.211,E2 -15524.211} C_VEL
LIN {X 0,Y 312.481,Z 205.558,A -85,B 0,C 180,E1 -15527.92,E2 -15527.92} C_VEL
LIN {X 0,Y 312.496,Z 205.561,A -85,B 0,C 180,E1 -15530.972,E2 -15530.972} C_VEL
LIN {X 0,Y 312.53,Z 205.555,A -85,B 0,C 180,E1 -15534.222,E2 -15534.222} C_VEL
LIN {X 0,Y 312.555,Z 205.743,A -85,B 0,C 180,E1 -15536.071,E2 -15536.071} C_VEL
LIN {X 0,Y 315.813,Z 220.174,A -85,B 0,C 180,E1 -15539.459,E2 -15539.459} C_VEL
LIN {X 0,Y 318.344,Z 231.562,A -85,B 0,C 180,E1 -15542.016,E2 -15542.016} C_VEL
LIN {X 0,Y 318.271,Z 235.006,A -85,B 0,C 180,E1 -15542.73,E2 -15542.73} C_VEL
LIN {X 0,Y 315.477,Z 258.293,A -85,B 0,C 180,E1 -15547.402,E2 -15547.402} C_VEL
LIN {X 0,Y 315.393,Z 259.524,A -85,B 0,C 180,E1 -15547.59,E2 -15547.59} C_VEL
LIN {X 0,Y 318.266,Z 293.555,A -85,B 0,C 180,E1 -15548.684,E2 -15548.684} C_VEL
LIN {X 0,Y 316.906,Z 364.563,A -85,B 0,C 180,E1 -15550.613,E2 -15550.613} C_VEL
LIN {X 0,Y 316.214,Z 377.264,A -85,B 0,C 180,E1 -15551.201,E2 -15551.201} C_VEL
LIN {X 0,Y 315.394,Z 389.057,A -85,B 0,C 180,E1 -15551.991,E2 -15551.991} C_VEL
LIN {X 0,Y 314.513,Z 401.44,A -85,B 0,C 180,E1 -15553.114,E2 -15553.114} C_VEL
LIN {X 0,Y 313.605,Z 412.449,A -85,B 0,C 180,E1 -15554.401,E2 -15554.401} C_VEL
LIN {X 0,Y 312.805,Z 421.342,A -85,B 0,C 180,E1 -15555.692,E2 -15555.692} C_VEL
LIN {X 0,Y 312.067,Z 430.466,A -85,B 0,C 180,E1 -15557.317,E2 -15557.317} C_VEL
LIN {X 0,Y 311.584,Z 437.944,A -85,B 0,C 180,E1 -15558.948,E2 -15558.948} C_VEL
LIN {X 0,Y 311.279,Z 445.183,A -85,B 0,C 180,E1 -15560.908,E2 -15560.908} C_VEL
LIN {X 0,Y 311.247,Z 450.863,A -85,B 0,C 180,E1 -15562.868,E2 -15562.868} C_VEL
LIN {X 0,Y 311.26,Z 455.199,A -85,B 0,C 180,E1 -15564.819,E2 -15564.819} C_VEL
LIN {X 0,Y 311.361,Z 457.446,A -85,B 0,C 180,E1 -15566.118,E2 -15566.118} C_VEL
LIN {X 0,Y 311.494,Z 459.146,A -85,B 0,C 180,E1 -15567.415,E2 -15567.415} C_VEL
LIN {X 0,Y 311.545,Z 460.372,A -85,B 0,C 180,E1 -15568.708,E2 -15568.708} C_VEL
LIN {X 0,Y 311.508,Z 461.145,A -85,B 0,C 180,E1 -15570.001,E2 -15570.001} C_VEL
LIN {X 0,Y 311.51,Z 461.43,A -85,B 0,C 180,E1 -15571.294,E2 -15571.294} C_VEL
LIN {X 0,Y 311.316,Z 461.265,A -85,B 0,C 180,E1 -15572.589,E2 -15572.589} C_VEL
LIN {X 0,Y 311.089,Z 460.675,A -85,B 0,C 180,E1 -15573.887,E2 -15573.887} C_VEL
LIN {X 0,Y 311.044,Z 458.543,A -85,B 0,C 180,E1 -15576.183,E2 -15576.183} C_VEL
LIN {X 0,Y 311.088,Z 455.078,A -85,B 0,C 180,E1 -15578.445,E2 -15578.445} C_VEL
LIN {X 0,Y 311.377,Z 450.925,A -85,B 0,C 180,E1 -15580.404,E2 -15580.404} C_VEL
LIN {X 0,Y 312.112,Z 445.626,A -85,B 0,C 180,E1 -15582.353,E2 -15582.353} C_VEL
LIN {X 0,Y 313.101,Z 439.009,A -85,B 0,C 180,E1 -15584.296,E2 -15584.296} C_VEL
LIN {X 0,Y 314.636,Z 430.487,A -85,B 0,C 180,E1 -15586.271,E2 -15586.271} C_VEL
LIN {X 0,Y 316.043,Z 422.353,A -85,B 0,C 180,E1 -15587.805,E2 -15587.805} C_VEL
LIN {X 0,Y 317.958,Z 412.105,A -85,B 0,C 180,E1 -15589.364,E2 -15589.364} C_VEL
LIN {X 0,Y 319.909,Z 400.602,A -85,B 0,C 180,E1 -15590.748,E2 -15590.748} C_VEL
LIN {X 0,Y 321.649,Z 389.413,A -85,B 0,C 180,E1 -15591.806,E2 -15591.806} C_VEL
LIN {X 0,Y 323.353,Z 376.795,A -85,B 0,C 180,E1 -15592.694,E2 -15592.694} C_VEL
LIN {X 0,Y 324.625,Z 363.711,A -85,B 0,C 180,E1 -15593.358,E2 -15593.358} C_VEL
LIN {X 0,Y 325.584,Z 344.511,A -85,B 0,C 180,E1 -15593.96,E2 -15593.96} C_VEL
LIN {X 0,Y 327.665,Z 297.369,A -85,B 0,C 180,E1 -15595.315,E2 -15595.315} C_VEL
LIN {X 0,Y 326.176,Z 280.603,A -85,B 0,C 180,E1 -15596.102,E2 -15596.102} C_VEL
LIN {X 0,Y 323.716,Z 264.61,A -85,B 0,C 180,E1 -15597.004,E2 -15597.004} C_VEL
LIN {X 0,Y 322.138,Z 255.387,A -85,B 0,C 180,E1 -15597.621,E2 -15597.621} C_VEL
LIN {X 0,Y 323.949,Z 244.609,A -85,B 0,C 180,E1 -15599.796,E2 -15599.796} C_VEL
LIN {X 0,Y 322.552,Z 236.896,A -85,B 0,C 180,E1 -15601.813,E2 -15601.813} C_VEL
LIN {X 0,Y 320.362,Z 227.984,A -85,B 0,C 180,E1 -15604.409,E2 -15604.409} C_VEL
LIN {X 0,Y 317.725,Z 219.607,A -85,B 0,C 180,E1 -15607.22,E2 -15607.22} C_VEL
LIN {X 0,Y 315.332,Z 213.119,A -85,B 0,C 180,E1 -15609.743,E2 -15609.743} C_VEL
LIN {X 0,Y 313.725,Z 208.786,A -85,B 0,C 180,E1 -15611.635,E2 -15611.635} C_VEL
LIN {X 0,Y 312.512,Z 205.666,A -85,B 0,C 180,E1 -15613.237,E2 -15613.237} C_VEL
LIN {X 0,Y 312.493,Z 205.558,A -85,B 0,C 180,E1 -15617.568,E2 -15617.568} C_VEL
LIN {X 0,Y 312.502,Z 205.56,A -85,B 0,C 180,E1 -15620.971,E2 -15620.971} C_VEL
LIN {X 0,Y 312.535,Z 205.55,A -85,B 0,C 180,E1 -15624.22,E2 -15624.22} C_VEL
LIN {X 0,Y 312.507,Z 205.558,A -85,B 0,C 180,E1 -15627.334,E2 -15627.334} C_VEL
LIN {X 0,Y 312.547,Z 205.55,A -85,B 0,C 180,E1 -15631.279,E2 -15631.279} C_VEL
LIN {X 0,Y 312.589,Z 205.545,A -85,B 0,C 180,E1 -15634.711,E2 -15634.711} C_VEL
LIN {X 0,Y 312.591,Z 205.545,A -85,B 0,C 180,E1 -15637.529,E2 -15637.529} C_VEL
LIN {X 0,Y 312.641,Z 205.541,A -85,B 0,C 180,E1 -15641.656,E2 -15641.656} C_VEL
LIN {X 0,Y 312.656,Z 205.742,A -85,B 0,C 180,E1 -15643.597,E2 -15643.597} C_VEL
LIN {X 0,Y 314.878,Z 211.465,A -85,B 0,C 180,E1 -15646.446,E2 -15646.446} C_VEL
LIN {X 0,Y 317.631,Z 219.568,A -85,B 0,C 180,E1 -15649.804,E2 -15649.804} C_VEL
LIN {X 0,Y 319.42,Z 225.353,A -85,B 0,C 180,E1 -15651.936,E2 -15651.936} C_VEL
LIN {X 0,Y 321.847,Z 235.678,A -85,B 0,C 180,E1 -15655.271,E2 -15655.271} C_VEL
LIN {X 0,Y 323.418,Z 239.714,A -85,B 0,C 180,E1 -15655.725,E2 -15655.725} C_VEL
LIN {X 0,Y 327.124,Z 254.933,A -85,B 0,C 180,E1 -15656.875,E2 -15656.875} C_VEL
LIN {X 0,Y 328.677,Z 262.672,A -85,B 0,C 180,E1 -15657.395,E2 -15657.395} C_VEL
LIN {X 0,Y 325.256,Z 322.924,A -85,B 0,C 180,E1 -15659.458,E2 -15659.458} C_VEL
LIN {X 0,Y 324.489,Z 334.741,A -85,B 0,C 180,E1 -15660.089,E2 -15660.089} C_VEL
LIN {X 0,Y 323.338,Z 346.787,A -85,B 0,C 180,E1 -15660.992,E2 -15660.992} C_VEL
LIN {X 0,Y 322.085,Z 357.228,A -85,B 0,C 180,E1 -15662.031,E2 -15662.031} C_VEL
LIN {X 0,Y 320.683,Z 367.135,A -85,B 0,C 180,E1 -15663.297,E2 -15663.297} C_VEL
LIN {X 0,Y 319.105,Z 376.098,A -85,B 0,C 180,E1 -15664.737,E2 -15664.737} C_VEL
LIN {X 0,Y 317.62,Z 384.07,A -85,B 0,C 180,E1 -15666.351,E2 -15666.351} C_VEL
LIN {X 0,Y 316.012,Z 391.567,A -85,B 0,C 180,E1 -15668.311,E2 -15668.311} C_VEL
LIN {X 0,Y 314.704,Z 397.196,A -85,B 0,C 180,E1 -15670.291,E2 -15670.291} C_VEL
LIN {X 0,Y 313.622,Z 401.321,A -85,B 0,C 180,E1 -15672.291,E2 -15672.291} C_VEL
LIN {X 0,Y 312.586,Z 404.493,A -85,B 0,C 180,E1 -15674.807,E2 -15674.807} C_VEL
LIN {X 0,Y 311.946,Z 405.609,A -85,B 0,C 180,E1 -15677.03,E2 -15677.03} C_VEL
LIN {X 0,Y 311.654,Z 405.446,A -85,B 0,C 180,E1 -15678.714,E2 -15678.714} C_VEL
LIN {X 0,Y 311.502,Z 404.908,A -85,B 0,C 180,E1 -15679.78,E2 -15679.78} C_VEL
LIN {X 0,Y 311.428,Z 403.644,A -85,B 0,C 180,E1 -15681.165,E2 -15681.165} C_VEL
LIN {X 0,Y 311.529,Z 400.611,A -85,B 0,C 180,E1 -15683.252,E2 -15683.252} C_VEL
LIN {X 0,Y 311.804,Z 396.022,A -85,B 0,C 180,E1 -15685.356,E2 -15685.356} C_VEL
LIN {X 0,Y 312.162,Z 390.828,A -85,B 0,C 180,E1 -15687.123,E2 -15687.123} C_VEL
LIN {X 0,Y 312.614,Z 383.513,A -85,B 0,C 180,E1 -15689.054,E2 -15689.054} C_VEL
LIN {X 0,Y 313.218,Z 375.561,A -85,B 0,C 180,E1 -15690.694,E2 -15690.694} C_VEL
LIN {X 0,Y 313.907,Z 366.185,A -85,B 0,C 180,E1 -15692.239,E2 -15692.239} C_VEL
LIN {X 0,Y 314.585,Z 356.013,A -85,B 0,C 180,E1 -15693.567,E2 -15693.567} C_VEL
LIN {X 0,Y 315.298,Z 344.155,A -85,B 0,C 180,E1 -15694.76,E2 -15694.76} C_VEL
LIN {X 0,Y 315.833,Z 332.36,A -85,B 0,C 180,E1 -15695.642,E2 -15695.642} C_VEL
LIN {X 0,Y 316.195,Z 320.26,A -85,B 0,C 180,E1 -15696.283,E2 -15696.283} C_VEL
LIN {X 0,Y 316.743,Z 295.961,A -85,B 0,C 180,E1 -15697.055,E2 -15697.055} C_VEL
LIN {X 0,Y 317.729,Z 253.908,A -85,B 0,C 180,E1 -15698.309,E2 -15698.309} C_VEL
LIN {X 0,Y 314.595,Z 232.033,A -85,B 0,C 180,E1 -15699.166,E2 -15699.166} C_VEL
LIN {X 0,Y 315.236,Z 220.86,A -85,B 0,C 180,E1 -15701.976,E2 -15701.976} C_VEL
LIN {X 0,Y 314.825,Z 217.133,A -85,B 0,C 180,E1 -15702.978,E2 -15702.978} C_VEL
LIN {X 0,Y 312.527,Z 205.692,A -85,B 0,C 180,E1 -15706.253,E2 -15706.253} C_VEL
LIN {X 0,Y 312.503,Z 205.56,A -85,B 0,C 180,E1 -15709.874,E2 -15709.874} C_VEL
LIN {X 0,Y 312.534,Z 205.554,A -85,B 0,C 180,E1 -15714.05,E2 -15714.05} C_VEL
LIN {X 0,Y 312.504,Z 205.558,A -85,B 0,C 180,E1 -15717.333,E2 -15717.333} C_VEL
LIN {X 0,Y 312.551,Z 205.553,A -85,B 0,C 180,E1 -15721.275,E2 -15721.275} C_VEL
LIN {X 0,Y 312.584,Z 205.545,A -85,B 0,C 180,E1 -15724.71,E2 -15724.71} C_VEL
